(* CODESYS project PMPS.library
   Author: Alex Wallace and contributors
   Placeholder: PMPS
   Description: Collection of PMPS functionality for LCLS PLCs
   Version: 0.0.0
   DefaultNamespace: PMPS
   Title: PMPS
   Company: SLAC - LCLS

Project tree, tasks and I/O mapping:
  libraries: LCLS General, * (SLAC); Tc2_MC2, * (Beckhoff Automation GmbH); Tc2_Standard, * (Beckhoff Automation GmbH); Tc2_System, * (Beckhoff Automation GmbH); Tc2_Utilities, * (Beckhoff Automation GmbH); Tc3_JsonXml, * (Beckhoff Automation GmbH); Tc3_Module, * (Beckhoff Automation GmbH); TcUnit, * (www.tcunit.org)
  DUTs/
    InternalDUT/
      data type E_BPTMState
      data type E_MPSBeamRates
      data type K_Apertures
      data type K_Stopper
      data type L_Apertures
      data type L_Stopper
      data type ST_FF
      data type ST_FFInfo
      data type ST_FFOverride
      data type ST_PMPS_Aperture
      data type ST_PMPS_Attenuator
      data type T_HashTableEntry
    UserDUT/
      data type ST_BeamParams
      data type ST_Device
    data type ST_DeviceState
    data type ST_DeviceStateExt
    data type ST_DeviceStateTable
  GVLs/
    global variables GVL_CUSTOM_CONSTANTS
    global variables PMPS_GVL
    global variables PMPS_TOOLS
  HelperFunctions/
    TypeTranslators/
      function APT_TO_IO [ST]
      function ATT_TO_IO [ST]
      function BP_TO_IO [ST]
      function F_DeviceState_To_DeviceStateExt [ST]
      function IO_TO_APT [ST]
      function IO_TO_ATT [ST]
      function IO_TO_BP [ST]
    function F_DifferentBeamParams [ST]
    function F_eVRangeCalculator [ST]
    function F_eVWithinSpec [ST]
    function F_PMPS_JSON [ST]
    function F_SafeBPCompare [ST]
    function F_SetBeamParams [ST]
    function F_SetStateParams [ST]
  MajorComponents/
    Arbiter/
      function block FB_Arbiter [ST]: AddRequest, ArbitrateBP, CheckRequest, CheckRequestInPool, ElevateRequest, FB_init, GetArbitratedBP, RemoveRequest, RequestBP
      function block FB_BeamParamAssertionPool [ST]: A_Add, A_Count, A_GetFirst, A_GetNext, A_Lookup, A_Remove, A_Reset
    FastFaults/
      function block FB_FastFault [ST]
      function block FB_HardwareFFOutput [ST]: EvaluateOutput, EvaluateOverrides, EvaluateVetos, Execute, ExecuteLogging, FormulateLogJson, IdxCheckIn, Register
    InterPlcComm/
      function block FB_ArbiterToSubSys_IO [ST]
      function block FB_SubSysToArbiter_IO [ST]: CheckRequest, RequestBP
    PhotonEnergyInterface/
      function F_CalculatePhotonEnergy [ST]
      function block FB_AcceleratorLinks [ST]
      function block FB_Hgvpu [ST]: Init, UndAdrUpdate
      function block FB_LPhotonEnergy [ST]
      function block FB_SXU [ST]
      function block FB_UndulatorSegment [ST]
    PMPS_MPS_Interface/
      function block FB_BeamClassOutputs [ST]
      function block FB_CTLS_Outputs [ST]
      function block FB_PhotonEnergyWatcher [ST]
    SimulationFB/
      function block FB_eVSimulator [ST]
      function block FB_MachineSimulator [ST]
    Stoppers/
      function block FB_KStopper [ST]: FB_init
      function block FB_LStopper [ST]: FB_init
      function block FB_StopperWatcher [ST]
    function block BeamParameterTransitionManager [ST]: AssertFinalBP, AssertTransitionBP, AuthorizeTransition, DeauthorizeTransition, NewTarget_ENTRY, RemoveTransitionAssertion, SetNewTarget, WaitingForFinalAssertion_DO, WaitingForFinalAssertion_EXIT, WaitingForTransitionAssertion_DO, WaitingForTransitionAssertion_EXIT
    function block FB_BPControlDevice [ST]: FB_init
    function block FB_BPRequestor [ST]: CheckRequest, RequestBP
    function block FB_LinearDeviceStateTable [ST]: A_Add, A_Count, A_GetFirst, A_GetNext, A_Lookup, A_Remove, A_Reset
    function block FB_LinearGovernor [ST]
    function block FB_LRateFromEPICS [ST]
    interface I_HigherAuthority: CheckRequest, RequestBP
  TestComponents/
    data type eBPTMTestStates
    function block FB_Arbiter_Test [ST]: Arbitration, FullArbitrationStack, RequestCheckRemoveBP, StackArbiters
    function block FB_ArbToSubsys_Test [ST]: BasicFunction
    function block FB_AttenuatorSimulator [ST]
    function block FB_BPTM_Test [ST]: BPTMBasicFunction
    function block FB_DiffBP_Test [ST]: BPDiff
    function block FB_evRangeCalculator_Test [ST]: BasicFunction
    function block FB_eVWithinSpec_Test [ST]: evWithinRangeChecks
    function block FB_FastFault_Test [ST]: FFCombinedFunctionality, FFRegistration
    function block FB_PhotonEnergyWatcher_Test [ST]: PEWatcherBasicFunction
    function block FB_SafeBPCompare_Test [ST]: BeamOffIsSafe, BPComparisonCheck
    function block FB_SubsysToArb_Test [ST]: BasicFunction
  VISUs/
  program MAIN [ST]
*)

// DUTs/InternalDUT/E_BPTMState
TYPE E_BPTMState :
(
    Init := 0,
	NewTarget := 1,
    WaitingForTransitionAssertion := 2,
    WaitingForFinalAssertion := 3,
    Transitioning := 4,
    CleaningUp := 5,
	Idle := 6
);
END_TYPE

// DUTs/InternalDUT/E_MPSBeamRates

TYPE E_MPSBeamRates :
(
	MPSRateInvalid            :=  0,
    MPSRate0Hz                :=  1,
    (* Previously used 2 and 3 for single shot and burst *)
    MPSRate1Hz                :=  4,
    MPSRate10Hz               :=  5,
    MPSRate30Hz               :=  6,
    MPSRate60Hz               :=  7,
    MPSRate120Hz              :=  8,
    MPSRateUnknown            :=  9,
    MPSRateSingleShot         := 10,
    MPSRateBurstMode          := 11,
    MPSRateBurstModeNotActive := 12,
    MPSNumberOfBeamRates      := 13,
    MPSRateBurstInvalid       := 14
)UINT;
END_TYPE

// DUTs/InternalDUT/K_Apertures
{attribute 'qualified_only'}
{attribute 'strict'}
TYPE K_Apertures :
(
	SL1K0 := 1,
    SL2K0 := 2
);
END_TYPE

// DUTs/InternalDUT/K_Stopper
{attribute 'qualified_only'}
{attribute 'strict'}
TYPE K_Stopper :
(
	ST1 := 1,
    ST2 := 2
);
END_TYPE

// DUTs/InternalDUT/L_Apertures
{attribute 'qualified_only'}
{attribute 'strict'}
TYPE L_Apertures :
(
	SL1L0 := 1,
    SL2L0 := 2
);
END_TYPE

// DUTs/InternalDUT/L_Stopper
{attribute 'qualified_only'}
{attribute 'strict'}
TYPE L_Stopper :
(
	ST1L0 := 1, // ST1
    ST1L1 := 2 // ST2
);
END_TYPE

// DUTs/InternalDUT/ST_FF
TYPE ST_FF :
STRUCT
    {attribute 'pytmc' := '
        pv: Info
     '}
    Info : ST_FFInfo;
    
    {attribute 'pytmc' := '
        pv: Ovrd
     '}
    Ovrd : ST_FFOverride;
    
    {attribute 'pytmc' := '
        pv: OK
        io: i
     '}
    OK   :   BOOL; // Fault logic state
    
    FaultAck : BOOL; // Set when faulted, reset by logger.
    ClearAck : BOOL;
    
    {attribute 'pytmc' := '
        pv: BeamPermitted
        io: i
     '}
    BeamPermitted   :   BOOL; // Result of reset, veto, and fault logic, true beam off boolean
    
    {attribute 'pytmc' := '
        pv: Reset
        io: o
     '}
    Reset   :   BOOL;
    
    bsFF    :    RS;
    rtReset    :    R_TRIG;
    ftCountFault : F_TRIG;
    
END_STRUCT
END_TYPE

// DUTs/InternalDUT/ST_FFInfo

// These elements should be set at init and never changed.

TYPE ST_FFInfo :
STRUCT
    {attribute 'pytmc' := '
        pv: Path
        io: i
     '}
    sPath   :    T_MaxString; // Full PLC path to FF object
    {attribute 'pytmc' := '
        pv: Desc
        io: i
     '}
    Desc    :   T_MaxString; // Set at instantiation to a helpful description of the fast fault purpose
    {attribute 'pytmc' := '
        pv: DevName
        io: i
     '}
    DevName :   T_MaxString; // Component name, used in diagnostic to help narrow down where beam faults are coming from
    {attribute 'pytmc' := '
        pv: TypeCode
        io: i
     '}
    TypeCode    :   UINT; // Set at instantiation to fault class code

///////////////////////////////////////////
// Warning, this variable is effectively a VETO of the fast fault if set FALSE
// Do not alter the state of this variable unless you really know what you're doing.
///////////////////////////////////////////
    {attribute 'pytmc' := '
        pv: InUse
        io: i
     '}
    InUse   :   BOOL := FALSE; // If this FF is currently in-use
///////////////////////////////////////////

 
    AutoReset   :   BOOL; // Automatically clear fast fault (latching vs non-latching)
    Vetoable  : BOOL := TRUE; // Can this fast fault be masked by the veto device input?

      {attribute 'pytmc' := '
        pv: InfoString
        io: i
     '}
    InfoString : STRING;
END_STRUCT
END_TYPE

// DUTs/InternalDUT/ST_FFOverride
TYPE ST_FFOverride :
STRUCT
    {attribute 'pytmc' := '
        pv: Duration
        io: o
     '}
    Duration : UDINT; // UDINT to be compatible with ESS module.
    
    {attribute 'pytmc' := '
        pv: Activate
        io: o
     '}
    Activate : BOOL;
    
    {attribute 'pytmc' := '
        pv: Deactivate
        io: o
     '}
    Deactivate : BOOL;
    
    {attribute 'pytmc' := '
        pv: ElapsedTime
        io: i
     '}
    ElapsedTime : UDINT; // UDINT to be compatible with ESS module.
    
    {attribute 'pytmc' := '
        pv: RemainingTime
        io: i
     '}
    RemainingTime : UDINT; // UDINT to be compatible with ESS module.
    
    {attribute 'pytmc' := '
        pv: Active
        io: i
     '} 
	Active: BOOL;
    
    Timer    :   TP;
    OvrdActLogAck : BOOL;
    OvrdExpLogAck : BOOL;
    
    tOvrdActivate : R_TRIG;
    tOvrdExpiring  : F_TRIG;
END_STRUCT
END_TYPE

// DUTs/InternalDUT/ST_PMPS_Aperture
TYPE ST_PMPS_Aperture EXTENDS ST_PMPS_Aperture_IO :
STRUCT
    (*
    {attribute 'pytmc' := 'pv: Width
            io: i
            field: EGU mm'}
    Width : REAL; // distance between horizontal slits (x)
    {attribute 'pytmc' := 'pv: Height
            io: i
            field: EGU mm'}
    Height : REAL; // distance between vertical slits (y)
    
    {attribute 'pytmc' := 'pv: OK
        io: i'}
    xOK : BOOL; // status of aperture, false if error or in motion
    *)
END_STRUCT
END_TYPE

// DUTs/InternalDUT/ST_PMPS_Attenuator
TYPE ST_PMPS_Attenuator EXTENDS ST_PMPS_Attenuator_IO :
STRUCT
    (*
        {attribute 'pytmc' := 'pv: Att
            io: i
            field: EGU %
        '}
		nTran : UINT;
        {attribute 'pytmc' := 'pv: OK
            io: i
        '}
		xAttOK : UINT; // true = no errors and attenuator is stable
        *)
END_STRUCT
END_TYPE

// DUTs/InternalDUT/T_HashTableEntry
TYPE T_HashTableEntry :
STRUCT
    {attribute 'pytmc' := '
        pv: Key
        io: i
     '}
    key : DWORD := 0;
    value : PVOID := 0;
END_STRUCT
END_TYPE

// DUTs/UserDUT/ST_BeamParams
TYPE ST_BeamParams : 
    STRUCT
        (*  Requested pre-optic attenuation %  *)
		{attribute 'pytmc' := 'pv: Transmission
            io: i
            field: EGU %
        '}
		nTran : UINT := 100;
        (* Pulse-rate *)
        {attribute 'pytmc' := 'pv: Rate
            io: i
            field: EGU Hz
        '}
        nRate : UDINT := 120;
        (* Per pulse max energy (mJ) *)
        {attribute 'pytmc' := 'pv: PulseEnergy
            io: i
            field: EGU mJ
            field: DESC This beam parameter is non-op for now.
        '}
        fPP_mJ : REAL := 20;
        (* Photon energy ranges *)
        {attribute 'pytmc' := 'pv: PhotonEnergyRanges
            io: i
            field: EGU eV'}
        {attribute 'displaymode' := 'binary'}
        neVRange : WORD := 2#1111_1111_1111_1111;
        (* Beamline attenuators *)
        {attribute 'pytmc' := 'pv: AuxAtt
        io: i'}
        astAttenuators : ARRAY [1..PMPS_GVL.AUX_ATTENUATORS] OF ST_PMPS_Attenuator;
        
        (* Stoppers *)
        {attribute 'pytmc' := 'pv: ST
        io: i'}
        aStoppers : ARRAY [1..PMPS_GVL.MAX_STOPPERS] OF BOOL;
        
        (* Apertures *)
        astApertures : ARRAY [1..PMPS_GVL.MAX_APERTURES] OF ST_PMPS_Aperture;
        
        // Toggle for watchdog
        xValidToggle : BOOL;
        // Beam parameter set is valid (if readback), or acknowledged (if request)
        {attribute 'pytmc' := 'pv: Valid
        io: i'}
        xValid : BOOL;
        // Cohort index. Identifies which cohort this BP set was included in arbitration
        {attribute 'pytmc' := 'pv: Cohort
        io: i
            field: DESC Cohort inc on each arb cycle
        '}
        nCohortInt : UDINT;
    END_STRUCT
END_TYPE

// DUTs/UserDUT/ST_Device
TYPE ST_Device :
STRUCT
	//IO
	stAxis	:	AXIS_REF;
	//The following limit switches must be TRUE or high (ie. NC) to enable that direction of motion
	//The EPICS display should show an inverted indicator to communicate end of travel reached
	i_xLoLim	AT %I*	:	BOOL; //Wire normally-closed
	i_xHiLim	AT %I*	:	BOOL; //Wire normally-closed
	
	//Acuator Parameters
	lrUpperPositionLimit	:	LREAL := 10000000000; //Use in conjuntion with limit switches or set to a huge number to ignore
	lrLowerPositionLimit	:	LREAL := -10000000000; //Use in conjuntion with limit switches or set to a huge number to ignore
	
	xEnable	:	BOOL := TRUE;
	
	//Supervisory System
	
	//MPS Override
	xOverrideMPSLimits	: BOOL := FALSE; //Set true to move beyond MPS limits. Note this will trip beam off.
	
	//Status and Faults
	xClearFaults	:	BOOL;	//Rising edge tries to clear faults of all kinds
	
	xGovernorFault	:	BOOL;	//Indicates governor is faulted
	xGovernorOverridden	:	BOOL; //Indicates governor is in override mode
	xSMFault		:	BOOL;	//Indicates component state machine is faulted
	
	//Device States
	StateTable		:	FB_LinearDeviceStateTable;
	
	stTransitionState	:	ST_DeviceState; //The transition state might have non-zero beam parameters
	nSafeState			:	UDINT; //State where the device is considered safe
	nTransitionState	:	UDINT;
	
	nRequestedState	:	UDINT; //EPICS control, cleaned (checked against array limits) and deposited in nTargetState
	nTargetState	:	UDINT; //The requested state should be deposited here after cleaning
	nActiveState	:	UDINT; //The last successfully reached state
	
	
END_STRUCT
END_TYPE

// DUTs/ST_DeviceState
TYPE ST_DeviceState :
STRUCT
	
	//State name
	sStateName	:	STRING;
	nStateRef	:	UDINT; //Primary key of device state database
	
	//////////////////
	// This stuff may belong in a sub-class or something
	//Position
	rPosition	:	REAL := 0; //Center of the state
	//Tolerance
	rTolerance :	REAL := 0; //+/- amount
	//////////////////
	//Required beam parameters
	stReqBeamParam	:	ST_BeamParams;

END_STRUCT
END_TYPE

// DUTs/ST_DeviceStateExt
//Use when working with states in code
//Extended with a valid boolean to indicate the structure was loaded
//properly
TYPE ST_DeviceStateExt EXTENDS ST_DeviceState :
STRUCT
	xValid	:	BOOL := FALSE;
END_STRUCT
END_TYPE

// DUTs/ST_DeviceStateTable
TYPE ST_DeviceStateTable :
STRUCT
	iDeviceID:DINT;
	iStateID:DINT;
	rTargetPosition: REAL;
	rTolerance: REAL;
	rTransmission: REAL;
	iBeamClass : DINT;
	iPulseRate: DINT;
	rPerPulseEnergy:REAL;
	rUpper_eV: REAL;
	rLower_eV: REAL;
	rPhotonEnergy: REAL;
END_STRUCT
END_TYPE

// TestComponents/eBPTMTestStates
{attribute 'qualified_only'}
{attribute 'strict'}
TYPE eBPTMTestStates :
(
    Init := 0,
    WaitingForValidID := 50,
    WaitingForTransitionAssertion := 100,
    WaitingForFinalAssertion    := 200,
    Transitioning    := 300,
    CleaningUp    := 400,
    AnotherState := 500
);
END_TYPE

// GVLs/GVL_CUSTOM_CONSTANTS
VAR_GLOBAL CONSTANT
    MAX_FAST_FAULTS : UINT := 50; // Maximum number of fast faults that can be associated with a FFO
END_VAR

// GVLs/PMPS_GVL
{attribute 'qualified_only'}
VAR_GLOBAL
    {attribute 'pytmc' := '
        pv: @(PREFIX)RequestedBP
        archive: 1Hz monitor
    '}
    stRequestedBeamParameters    :    ST_BeamParams; //Summarized request for the line, as recognized by the line arbiter PLC
    {attribute 'pytmc' := '
        pv: @(PREFIX)CurrentBP
        archive: 1Hz monitor
    '}
    stCurrentBeamParameters    :    ST_BeamParams; //Currently active BP set, broadcast by the line arbiter PLC
    
    fbLog : FB_LogMessage:=(eSubsystem:=E_Subsystem.MPS);
END_VAR
VAR_GLOBAL RETAIN    
    // Statistics
    {attribute 'pytmc' := '
        pv: @(PREFIX)SuccessfulPreemptions
        io: i
    '}
    SuccessfulPreemption : UDINT; // Any time BPTM applies a new BP request which is confirmed
    {attribute 'pytmc' := '
        pv: @(PREFIX)AccumulatedFastFaults
        io: i
    '}
    AccumulatedFF : UDINT; // Any time a FF occurs
END_VAR
VAR_GLOBAL CONSTANT
    EXCLUDED_ASSERTION_ID    :    UDINT    := 16#FFFFFFFF; //An assertion ID that should always return "not found" in the assertion pool
    VISIBLE_TEST_VELOCITY    :    LREAL    := 10;
    FAST_TEST_VELOCITY        :    LREAL    := 100;
    MAX_DEVICE_STATES        :    UDINT    := 300;

    MAX_STOPPERS    :   UINT := 16;
    {attribute 'pytmc' := '
        pv: @(PREFIX)FullBeamCnst
        archive: 1Hz monitor
        field: DESC Full beam constant
    '}    
    cstFullBeam    :    ST_BeamParams := (
        nTran := 100,
        fPP_mJ := 1E4,
        neVRange := 2#1111_1111_1111_1111,
        nRate    := UDINT#1000000
    );
    {attribute 'pytmc' := '
        pv: @(PREFIX)SafeBeamCnst
        archive: 1Hz monitor
        field: DESC Safe beam constant
    '} 
    cstSafeBeam    :    ST_BeamParams := (
        nTran := 0,
        fPP_mJ := 0,
        neVRange := 0,
        nRate    := 0
    );
    
    cnMaxStateArrayLen : INT := 20;
    
    AUX_ATTENUATORS : UINT := 16; // Maximum # of attenuators in the PMPS
    MAX_APERTURES : UINT := 4; // Maximum # of power slits in the PMPS
    {warning disable C0228}
    DUMMY_AUX_ATT_ARRAY : ARRAY [1..PMPS_GVL.AUX_ATTENUATORS] OF ST_PMPS_Attenuator;
    {warning restore C0228}
    MAX_ASSERTIONS    :    UDINT := 20; //Maximum number of assertions permitted in the arbiter
    
    g_cBoundaries    :    INT    := 15;
    {attribute 'pytmc' := '
        pv: @(PREFIX)eVRangeHyst
        archive: 1Hz monitor
        field: DESC eV Range hystersis
        field: EGU eV
    '}
    reVHyst: REAL := 5; // 
    {attribute 'pytmc' := '
        pv: @(PREFIX)eVRangeCnst
        archive: 1Hz monitor
        field: DESC eV Range constants
        field: EGU eV
    '}
    g_areVBoundaries    :    ARRAY [0..g_cBoundaries]    OF    REAL    := [
    1E3,
    2.7E3,
    4.4E3,
    6.1E3,
    7.8E3,
    9.5E3,
    11.2E3,
    12.9E3,
    14.6E3,
    16.3E3,
    18E3,
    19.7E3,
    21.4E3,
    23.1E3,
    24.8E3,
    25E3
];


//////////////////////////
// Undulator constants
//////////////////////////
    {attribute 'pytmc' := '
		pv: @(PREFIX)L:UND:FirstSegment 
		io: i
	'}
    iLowBound_LUnd  : UDINT := 24;
    {attribute 'pytmc' := '
		pv: @(PREFIX)L:UND:LastSegment
		io: i
	'}
    iHighBound_LUnd : UDINT := 46;
    {attribute 'pytmc' := '
        pv: Period
        io: i
        field: EGU mm
    '}
    fPeriod_mm_LUnd : LREAL := 26.0;
	{attribute 'pytmc' := '
        pv: @(PREFIX)L:UND:LowK
        io: i
    '}
	fLowK_LUnd : LREAL := 0.54;
	{attribute 'pytmc' := '
        pv: @(PREFIX)L:UND:HiK
        io: i
    '}
	fHiK_LUnd : LREAL := 2.5;

END_VAR

// GVLs/PMPS_TOOLS
{attribute 'qualified_only'}
VAR_GLOBAL
	fbJson : FB_JsonSaxWriter;
END_VAR

// HelperFunctions/TypeTranslators/APT_TO_IO
FUNCTION APT_TO_IO : ST_PMPS_Aperture_IO
VAR_INPUT
    Apt : ST_PMPS_Aperture;
END_VAR
VAR
END_VAR

APT_TO_IO.Height := Apt.Height;
APT_TO_IO.Width := Apt.Width;
APT_TO_IO.xOK := Apt.xOK;

END_FUNCTION

// HelperFunctions/TypeTranslators/ATT_TO_IO
FUNCTION ATT_TO_IO : ST_PMPS_Attenuator_IO
VAR_INPUT
    Att : ST_PMPS_Attenuator;
END_VAR
VAR
END_VAR

ATT_TO_IO.nTran := Att.nTran;
ATT_TO_IO.xAttOK := Att.xAttOK;

END_FUNCTION

// HelperFunctions/TypeTranslators/BP_TO_IO
FUNCTION BP_TO_IO : ST_BeamParams_IO
VAR_INPUT
    BP : ST_BeamParams;
END_VAR
VAR
    idx : UINT := 0;
END_VAR


FOR idx := 1 TO PMPS_GVL.AUX_ATTENUATORS DO
    BP_TO_IO.astAttenuators[idx] := ATT_TO_IO(BP.astAttenuators[idx]);
END_FOR

FOR idx := 1 TO PMPS_GVL.MAX_APERTURES DO
    BP_TO_IO.astApertures[idx] := APT_TO_IO(BP.astApertures[idx]);
END_FOR

BP_TO_IO.aStoppers := BP.aStoppers;
BP_TO_IO.nTran := BP.nTran;
BP_TO_IO.fPP_mJ := BP.fPP_mJ;
BP_TO_IO.nCohortInt := ULINT_TO_UDINT(BP.nCohortInt);
BP_TO_IO.neVRange := BP.neVRange;
BP_TO_IO.nRate := BP.nRate;
BP_TO_IO.xValid := BP.xValid;
BP_TO_IO.xValidToggle := BP.xValidToggle;

END_FUNCTION

// HelperFunctions/TypeTranslators/F_DeviceState_To_DeviceStateExt
FUNCTION F_DeviceState_To_DeviceStateExt : ST_DeviceStateExt
VAR_INPUT
    stDeviceState    :    ST_DeviceState;
    xValid    :    BOOL;
END_VAR
VAR
END_VAR

F_DeviceState_To_DeviceStateExt.nStateRef := stDeviceState.nStateRef;
F_DeviceState_To_DeviceStateExt.rPosition    :=    stDeviceState.rPosition;
F_DeviceState_To_DeviceStateExt.rTolerance    :=    stDeviceState.rTolerance;
F_DeviceState_To_DeviceStateExt.sStateName    := stDeviceState.sStateName;
F_DeviceState_To_DeviceStateExt.stReqBeamParam    := stDeviceState.stReqBeamParam;
F_DeviceState_To_DeviceStateExt.xValid := xValid;

END_FUNCTION

// HelperFunctions/TypeTranslators/IO_TO_APT
FUNCTION IO_TO_APT : ST_PMPS_Aperture
VAR_INPUT
    IO : ST_PMPS_Aperture_IO;
END_VAR
VAR
END_VAR

IO_TO_APT.Height := IO.Height;
IO_TO_APT.Width := IO.Width;
IO_TO_APT.xOK := IO.xOK;

END_FUNCTION

// HelperFunctions/TypeTranslators/IO_TO_ATT
FUNCTION IO_TO_ATT : ST_PMPS_Attenuator
VAR_INPUT
    IO : ST_PMPS_Attenuator_IO;
END_VAR
VAR
END_VAR

IO_TO_ATT.nTran := IO.nTran;
IO_TO_ATT.xAttOK := IO.xAttOK;

END_FUNCTION

// HelperFunctions/TypeTranslators/IO_TO_BP
FUNCTION IO_TO_BP : ST_BeamParams
VAR_INPUT
    IO : ST_BeamParams_IO;
END_VAR
VAR
    idx : UINT;
END_VAR


FOR idx := 1 TO PMPS_GVL.AUX_ATTENUATORS DO
    IO_TO_BP.astAttenuators[idx] := IO_TO_ATT(IO.astAttenuators[idx]);
END_FOR

FOR idx := 1 TO PMPS_GVL.MAX_APERTURES DO
    IO_TO_BP.astApertures[idx] := IO_TO_APT(IO.astApertures[idx]);
END_FOR

IO_TO_BP.aStoppers := IO.aStoppers;
IO_TO_BP.nTran := IO.nTran;
IO_TO_BP.fPP_mJ := IO.fPP_mJ;
IO_TO_BP.nCohortInt := ULINT_TO_UDINT(IO.nCohortInt);
IO_TO_BP.neVRange := IO.neVRange;
IO_TO_BP.nRate := IO.nRate;
IO_TO_BP.xValid := IO.xValid;
IO_TO_BP.xValidToggle := IO.xValidToggle;

END_FUNCTION

// HelperFunctions/F_DifferentBeamParams
(*Compares BeamParam1 to BeamParam2, if any parameters of BeamParam1 are different than BeamParam2
the result will be true. *)
FUNCTION F_DifferentBeamParams : BOOL
VAR_INPUT
    BeamParam1    :    ST_BeamParams;
    BeamParam2    :    ST_BeamParams;
END_VAR
VAR
    xAttOK: BOOL := FALSE;
    xPPmjOK: BOOL := FALSE;
    xEvOK: BOOL := FALSE;
    xRateOK: BOOL := FALSE;
    xaStopper : BOOL := FALSE;
    xaAtt : BOOL := FALSE;
    xaApt : BOOL := FALSE;
    
    idx : UINT;
    
    
END_VAR

xAttOK := BeamParam1.nTran <> BeamParam2.nTran;
xPPmjOK := BeamParam1.fPP_mJ <> BeamParam2.fPP_mJ;
xEvOK := BeamParam1.neVRange <> BeamParam2.neVRange;
xRateOK     := BeamParam1.nRate <> BeamParam2.nRate;

//ast Attenuators
FOR idx:=1 TO PMPS_GVL.AUX_ATTENUATORS DO
    xaAtt S= (BeamParam1.astAttenuators[idx].nTran <> BeamParam2.astAttenuators[idx].nTran);   
END_FOR

// Stoppers
FOR idx:=1 TO PMPS_GVL.MAX_STOPPERS DO
    xaStopper S= (BeamParam1.aStoppers[idx] <> BeamParam2.aStoppers[idx]);
END_FOR

// ast Apertures
FOR idx:=1 TO PMPS_GVL.MAX_APERTURES DO
    xaApt S= (BeamParam1.astApertures[idx].Height <> BeamParam2.astApertures[idx].Height) OR
            (BeamParam1.astApertures[idx].Width <> BeamParam2.astApertures[idx].Width);
END_FOR


F_DifferentBeamParams := xAttOK OR xPPmjOK OR xEvOK OR xRateOK OR xaStopper OR xaAtt OR xaApt;

END_FUNCTION

// HelperFunctions/F_eVRangeCalculator
(*
A. Wallace 2019-8-8

Provides bit range of eV.

LastWord = 0 (Result)
----------------------------------
reV = 300 = (0000_0000_0000_0010)
reV = 301 = (0000_0000_0000_0100)

LastWord = 0000_0000_0000_0010 (Result)
----------------------------------
reV = 300 + <rHyst = (0000_0000_0000_0110)
reV = 300 + >rHyst = (0000_0000_0000_0100)

*)
FUNCTION F_eVRangeCalculator : WORD // Bit-range of current photon energy
VAR_INPUT
    reV    :    REAL; // Photon energy (keV)
    LastWord    :    WORD; // Range word of previous cycle
END_VAR
VAR
    nIndex: INT;
    RangeWord: WORD;
    rPreviousBoundary: REAL := 0;
    
    MaxEv    :    REAL := PMPS_GVL.g_areVBoundaries[PMPS_GVL.g_cBoundaries]*1000;
END_VAR


IF reV < 0 THEN F_eVRangeCalculator := 16#FFFF; RETURN; END_IF // Failsafe

FOR nIndex := 0 TO PMPS_GVL.g_cBoundaries DO
    
    // If previously active then check if it should be cleared
    IF LastWord.0 THEN 
        // Hysteresis condition
        IF (reV > MIN(PMPS_GVL.g_areVBoundaries[nIndex] + PMPS_GVL.reVHyst, MaxEv) ) OR
        (reV < MAX(rPreviousBoundary - PMPS_GVL.reVHyst, 0) ) THEN
            RangeWord.0 := 0; // If out of range of hys. mark inactive
        ELSE
            RangeWord.0 := 1;
        END_IF
    ELSE // Check if we should mark as active
        IF (reV <= PMPS_GVL.g_areVBoundaries[nIndex]) AND
        (reV > rPreviousBoundary) THEN
            RangeWord.0 := 1;
        END_IF
    END_IF
    
    // Catch if the hysteresis is set too large for the range
    IF rPreviousBoundary + PMPS_GVL.reVHyst >= PMPS_GVL.g_areVBoundaries[nIndex] THEN
        RangeWord.0 := 1; // Setting the bit true here as a failsafe
        //<TODO> Add major error or warning here
    END_IF
    
    rPreviousBoundary := PMPS_GVL.g_areVBoundaries[nIndex];
    // Shift to next bit
    RangeWord := ROR(RangeWord, 1);
    LastWord := SHR(LastWord, 1);
    
END_FOR

F_eVRangeCalculator := RangeWord;

END_FUNCTION

// HelperFunctions/F_eVWithinSpec
//reV must be within permitted range.
FUNCTION F_eVWithinSpec : BOOL
VAR_INPUT
    reV    :    REAL;    //Photon energy to check if within permitted range
    nPermittedRange    :    WORD; //Permitted range
END_VAR
VAR
    //Holding register for permitted ranges
    nPermittedRangeHolding    :    WORD; 
    //For loop counter
    nIndex    :    INT;
    // Lower boundary for range check 
    rPreviousBoundary: REAL := 0;
END_VAR

(* How this works:
The within range bool is initialized to false.
Load the word representation of ranges into a holding register.
If the bit at position zero of the holding register is true, and the input eV is
below the boundary at the index position of the boundary array, and the previous boundary
(which initializes at 0), then the within range bool is set. 
Then, we stash the upper boundary as the lower boundary for the next comparison,
and shift the holding register right, which moves the next bit to the zero position.
*)
nPermittedRangeHolding := nPermittedRange;

FOR nIndex := 0 TO PMPS_GVL.g_cBoundaries DO
        
    F_eVWithinSpec S= nPermittedRangeHolding.0 AND( 
        (reV <= PMPS_GVL.g_areVBoundaries[nIndex]*1000) AND
        (reV >= rPreviousBoundary*1000) );
        
    IF F_eVWithinSpec THEN RETURN; END_IF
    
    rPreviousBoundary := PMPS_GVL.g_areVBoundaries[nIndex];
    nPermittedRangeHolding := SHR(nPermittedRangeHolding, 1);
END_FOR

END_FUNCTION

// HelperFunctions/F_PMPS_JSON
FUNCTION F_PMPS_JSON : STRING
VAR_INPUT
	sDevName : STRING := '';
	sPath : STRING := '';
	nTypeCode : UINT := 0;
END_VAR
VAR
	
END_VAR


PMPS_TOOLS.fbJson.StartObject();
PMPS_TOOLS.fbJson.AddKey('pmps_typecode');
PMPS_TOOLS.fbJson.AddUdint(nTypeCode);
PMPS_TOOLS.fbJson.AddKey('pmps_path');
PMPS_TOOLS.fbJson.AddString(sPath);
PMPS_TOOLS.fbJson.AddKey('pmps_device_name');
PMPS_TOOLS.fbJson.AddString(sDevName);
PMPS_TOOLS.fbJson.EndObject();
F_PMPS_JSON := PMPS_TOOLS.fbJson.GetDocument();
PMPS_TOOLS.fbJson.ResetDocument();

END_FUNCTION

// HelperFunctions/F_SafeBPCompare
(*Compares BeamParam1 to BeamParam2: if the parameters of BeamParam1 are more conservative than BeamParam2
the result will be true. *)
FUNCTION F_SafeBPCompare : BOOL
VAR_INPUT
    BeamParam1    :    ST_BeamParams; //Must be more conservative than 2
    BeamParam2    :    ST_BeamParams;
END_VAR
VAR
    // Internal Attenuation OK boolean
    xAttOK: BOOL := FALSE;
    // Internal Per-pulse energy OK boolean
    xPPmjOK: BOOL := FALSE;
    // Internal photon energy OK boolean
    xEvOK: BOOL := FALSE;
    // Internal Beam Rate OK boolean
    xRateOK: BOOL;
    // Beam-rate is zero, masks all others considerations.
    xZeroRate: BOOL;
    
    idx : UINT;
    xAuxAttOK : BOOL := TRUE;
    xAuxAprtOK : BOOL := TRUE; 
END_VAR


xAttOK := BeamParam1.nTran <= BeamParam2.nTran;
xPPmjOK := BeamParam1.fPP_mJ <= BeamParam2.fPP_mJ;
xEvOK := (BeamParam1.neVRange AND BeamParam2.neVRange) = BeamParam1.neVRange;
xZeroRate    := BeamParam1.nRate = 0;
xRateOK    := BeamParam1.nRate <= BeamParam2.nRate;

FOR idx:=1 to PMPS_GVL.AUX_ATTENUATORS DO
    xAuxAttOK R= BeamParam1.astAttenuators[idx].nTran > BeamParam2.astAttenuators[idx].nTran;    
END_FOR

FOR idx:=1 to PMPS_GVL.MAX_APERTURES DO
    xAuxAprtOK R= BeamParam1.astApertures[idx].Height > BeamParam2.astApertures[idx].Height OR
    BeamParam1.astApertures[idx].Width > BeamParam2.astApertures[idx].Width;
END_FOR

F_SafeBPCompare := xZeroRate OR (xAttOK AND xPPmjOK AND xEvOK AND xRateOK AND xAuxAprtOK AND xAuxAttOK);

END_FUNCTION

// HelperFunctions/F_SetBeamParams
FUNCTION F_SetBeamParams : ST_BeamParams
VAR_INPUT
    nTran    :    UINT := 0;
    fPP_mJ: REAL := 0;
    neVRange    :    WORD := 0;
    nRate    :    UDINT := 0;
    astAuxAtt : ARRAY [1..PMPS_GVL.AUX_ATTENUATORS] OF ST_PMPS_Attenuator;
END_VAR
VAR
    BeamParams    :    ST_BeamParams;
    
END_VAR

BeamParams.nTran := LIMIT(0,nTran,100);
BeamParams.astAttenuators := astAuxAtt;
BeamParams.fPP_mJ := LIMIT(0,fPP_mJ,20);
BeamParams.neVRange := neVRange;
BeamParams.nRate    := MIN(nRate,1000000);

F_SetBeamParams    := BeamParams;

END_FUNCTION

// HelperFunctions/F_SetStateParams
FUNCTION F_SetStateParams : BOOL;
VAR_INPUT
    nStateRef    :    UDINT;
    rPosition    :    REAL;
    rTolerance: REAL;
    stBeamParams    :    ST_BeamParams;
END_VAR
VAR_IN_OUT
    Table    :    FB_LinearDeviceStateTable;
END_VAR
VAR
    stDeviceState    :    ST_DeviceState;
    
END_VAR

stDeviceState.nStateRef := nStateRef;
stDeviceState.rPosition := rPosition;
stDeviceState.rTolerance := rTolerance;
stDeviceState.stReqBeamParam := stBeamParams;

Table.A_Add(
    key := nStateRef,
    putValue := stDeviceState
);

F_SetStateParams := Table.bOk;

END_FUNCTION

// MajorComponents/FB_LinearDeviceStateTable
(* This function block implements simple database. Data element values are stored in the hash table.  *)
FUNCTION_BLOCK FB_LinearDeviceStateTable
VAR_INPUT
    key         : DWORD := 0;(* Entry key: used by A_Lookup, A_Remove method, the key variable is also used by A_Add method *)
    putPosPtr    : POINTER TO T_HashTableEntry := 0;(* Hash table entry position pointer (used by A_Find, A_GetNext, A_GetPrev) *)
    putValue     : ST_DeviceState;(* Hash table entry value (used by A_AddHead, A_AddTail, A_Find )*)
END_VAR
VAR_OUTPUT
    bOk            : BOOL := FALSE;(* TRUE = Success, FALSE = Failed *)
    getPosPtr    : POINTER TO T_HashTableEntry := 0;(* Returned hash table entry position pointer *)
    getValue     : ST_DeviceState;(* Returned hash table entry value *)
    nCount        : UDINT := 0;(* Hash table size (number of used entries, used by A_Count) *)
END_VAR
VAR
    dataPool    : ARRAY[0..PMPS_GVL.MAX_DEVICE_STATES] OF ST_DeviceState;(* Structured data element pool *)
    entries        : ARRAY[0..PMPS_GVL.MAX_DEVICE_STATES] OF T_HashTableEntry;(* Max. number of hash table entries. The value of table entry = 32 bit integer (pointer to dataPool-array-entry) *)
    fbTable     : FB_HashTableCtrl;(* basic hash table control function block *)
    hTable         : T_HHASHTABLE;(* hash table handle *)
    pRefPtr        : POINTER TO ST_DeviceState := 0;
    indexOfElem    : ULINT;(* Integer value (max. size: x86=>32bit, x64=>64bit)*)
END_VAR

;

ACTION A_Add:
(* Adds entry to the table *)
MEMSET( ADR( getValue ), 0, SIZEOF( getValue ) );
getPosPtr := 0;

fbTable.A_Add( hTable := hTable, key := key, putValue := ADR(PMPS_GVL.cstSafeBeam)(* we will set this value later *), getPosPtr=>getPosPtr, bOk=>bOk );(* Add new element to the table, getPosPtr points to the new entry *)
IF fbTable.bOk THEN(* Success *)
    fbTable.A_GetIndexAtPosPtr( hTable := hTable, putPosPtr := getPosPtr, getValue =>indexOfElem, bOk=>bOk );(* Get array index of getPosPtr entry *)
    IF fbTable.bOk THEN(* Success *)
        pRefPtr     := ADR( dataPool[indexOfElem] );(* Get pointer to the data element *)

        pRefPtr^ := putValue;(* copy application value *)

        fbTable.A_Add( hTable := hTable, key := key, putValue := pRefPtr, bOk=>bOk );(* Assign the entry value = pointer to the data element *)
        IF fbTable.bOk THEN(* Success *)
            getValue := putValue;
        END_IF
    END_IF
END_IF
END_ACTION

ACTION A_Count:
(* Count number of used entries *)
nCount := hTable.nCount;
bOk := TRUE;
END_ACTION

ACTION A_GetFirst:
(* Get first entry position pointer and value *)
MEMSET( ADR( getValue ), 0, SIZEOF( getValue ) );
getPosPtr := 0;

fbTable.A_GetFirst( hTable := hTable, putPosPtr := putPosPtr, getValue=>pRefPtr, getPosPtr=>getPosPtr, bOk=>bOk );
IF fbTable.bOk THEN
    getValue := pRefPtr^;
END_IF
END_ACTION

ACTION A_GetNext:
(* Get next entry position pointer and value *)
MEMSET( ADR( getValue ), 0, SIZEOF( getValue ) );
getPosPtr := 0;
bOk := FALSE;

IF putPosPtr = 0 THEN
    RETURN;
END_IF

fbTable.A_GetNext( hTable := hTable, putPosPtr := putPosPtr, getValue=>pRefPtr, getPosPtr=>getPosPtr, bOk=>bOk );
IF fbTable.bOk THEN
    getValue := pRefPtr^;
END_IF
END_ACTION

ACTION A_Lookup:
(* Lookup for entry by key  *)
MEMSET( ADR( getValue ), 0, SIZEOF( getValue ) );
getPosPtr := 0;

fbTable.A_Lookup( key := key, hTable := hTable, putPosPtr := putPosPtr, getValue=>pRefPtr, getPosPtr=>getPosPtr, bOk=>bOk );
IF fbTable.bOk THEN
    getValue := pRefPtr^;
END_IF
END_ACTION

ACTION A_Remove:
(* Search for entry and remove it *)
MEMSET( ADR( getValue ), 0, SIZEOF( getValue ) );
getPosPtr := 0;

fbTable.A_Remove( key := key, hTable := hTable, putPosPtr := putPosPtr, getValue=>pRefPtr, getPosPtr=>getPosPtr, bOk=>bOk );
IF fbTable.bOk THEN
    getValue := pRefPtr^;
END_IF
END_ACTION

ACTION A_Reset:
(* Reset/initialize linked list *)
MEMSET( ADR( getValue ), 0, SIZEOF( getValue ) );
getPosPtr := 0;
bOk := F_CreateHashTableHnd( ADR( entries ), SIZEOF( entries ), hTable );(* Intialize table handle *)
fbTable.A_Reset( hTable := hTable, bOk=>bOk );
nCount := 0;
END_ACTION

END_FUNCTION_BLOCK

// MajorComponents/Arbiter/FB_Arbiter
(* FB Arbiter
A. Wallace 2020-6-26

The arbiter primary objectives are:
- Provide a simple interface for devices to request beam parameter sets
- Provide a way for devices to verify their BPS is active in the arbiter
- Provide a way for devices remove their requests from evaluation
- Evaluate all active beam parameter requests registered with the aribiter,
to determine the safest combination of all sets, provide this set as an output.
- Do all of this with minimal overhead

To these ends, the arbiter uses a hash-table, the rows being a state-id as the key, and a corresponding
 beam parameter set to be evaluated against all the other sets (or rows), in the table.
 
The hash table can be thought of as an array on steriods, they are worth reading about, suffice to say
the hash table will tell you when you reach the end of all the entries, and enables us to find entries quickly.

These features efficiently address the addition, removal, and verification of beam parameter sets listed in the above requirements.
*)

FUNCTION_BLOCK FB_Arbiter IMPLEMENTS I_HigherAuthority
VAR_INPUT
END_VAR
VAR_OUTPUT
    {attribute 'pytmc' := '
        pv: ArbitratedBP
        io: i
        field: DESC Arbitrated BP
     '}
    q_stBeamParams    :    ST_BeamParams; //Updated on each cycle of the arbiter FB with the current arbitrated beam parameter set
    
    q_xStateIDFound    :    BOOL; //Set true if a state-id is found in the assertion pool after calling A_VerifyAssertion
END_VAR
VAR
    {attribute 'pytmc' := '
        pv: AP
        io: i
        field: DESC Assertion Pool
     '}
    fbBPAssertionPool    :    FB_BeamParamAssertionPool; //Table of active beam parameter assertions

    xRequestMade : BOOL; // Arbiter has confirmed its request has made it into the beam parameter request    
    
    {attribute 'pytmc' := '
        pv: ArbiterID
        io: i
        field: DESC Arbiter ID for elev. req.
     '}
    nArbiterID : UDINT; // Arbiter ID, used for making higher-level BP requests
    {attribute 'pytmc' := '
        pv: CohortCounter
        io: i
        field: DESC Intrnl cohort counter
     '}
    nArbiterCohort : UDINT := 1; // The cohort index keeps track of which beam parameter requests have been included in higher-level arbitrations
    // Init to 1, provides a guard against default cohort value in BP requests.
    {attribute 'pytmc' := '
        pv: ActiveInArbitration
        io: i
        field: DESC True if this arbiter's req is included
     '}
    xActiveInArbitration : BOOL; // True when this arbiter's request is included in all higher-level arbitrations
	
	nEntryCount : UDINT;
END_VAR

// Adds a request to the arbiter pool.
// Returns true if the request was successfully added, false if not enough space or a request with the same ID is already present.
METHOD AddRequest : BOOL
VAR_INPUT
    nReqID    :    DWORD; // Unique ID within aribter for the request. Make sure this is unique for every device + state combination
    stReqBP        :    ST_BeamParams; //Requested beam params
END_VAR
VAR_INST
    fbLog : FB_LogMessage;
END_VAR
// If the request is already in the pool, then skip the rest.
// This is flawed, needs to update the request if it's already in the pool, despite having the same ID
IF THIS^.CheckRequestInPool(nReqID) THEN
    AddRequest := FALSE;
    RETURN;
END_IF

IF nReqID <> PMPS_GVL.EXCLUDED_ASSERTION_ID THEN
    stReqBP.nCohortInt := nArbiterCohort; // Set the cohort number for this BP request.
    
    THIS^.fbBPAssertionPool.A_Add(
        key := nReqID,
        putValue := stReqBP
    );
END_IF
    
IF NOT THIS^.fbBPAssertionPool.bOk THEN
    fbLog(sMsg:=CONCAT(DWORD_TO_STRING(nReqID),'Addition to arbiter assertion pool failed'),
            eSevr:=TcEventSeverity.Warning,
            eSubsystem:=E_Subsystem.MPS);
ELSIF THIS^.fbBPAssertionPool.bOk THEN
	fbLog(sMsg:=CONCAT(DWORD_TO_STRING(nReqID),'Added to pool'),
            eSevr:=TcEventSeverity.Verbose,
            eSubsystem:=E_Subsystem.MPS);
END_IF

// With any new request reset the internal arbiter "done" flag
xRequestMade R= THIS^.fbBPAssertionPool.bOk;

AddRequest := THIS^.fbBPAssertionPool.bOk;
END_METHOD

// Kernel of the arbiter
// Logic for determining which beam parameter is the most conservative across all request sets.
METHOD INTERNAL ArbitrateBP : ST_BeamParams
VAR_INPUT
    stBP1    :    ST_BeamParams;
    stBP2    :    ST_BeamParams;
END_VAR
VAR
    idx : UINT := 1;
END_VAR
//<TODO>Add something here to register the key that won for each param

//Attenuation
ArbitrateBP.nTran := MIN(stBP1.nTran, stBP2.nTran);

FOR idx := 1 TO PMPS_GVL.AUX_ATTENUATORS DO
    ArbitrateBP.astAttenuators[idx].nTran := MIN(stBP1.astAttenuators[idx].nTran, stBP2.astAttenuators[idx].nTran);
END_FOR

//Apertures
FOR idx := 1 TO PMPS_GVL.MAX_APERTURES DO
    ArbitrateBP.astApertures[idx].Height := MIN(stBP1.astApertures[idx].Height, stBP2.astApertures[idx].Height);
    ArbitrateBP.astApertures[idx].Width := MIN(stBP1.astApertures[idx].Width, stBP2.astApertures[idx].Width);
END_FOR

//Pulse energy
ArbitrateBP.fPP_mJ := MIN(stBP1.fPP_mJ, stBP2.fPP_mJ);

//Photon energy ranges
ArbitrateBP.neVRange := stBP1.neVRange AND stBP2.neVRange;

//Rate
ArbitrateBP.nRate := MIN(stBP1.nRate, stBP2.nRate);
END_METHOD

(* Checks request ID is included in arbitration all the way to the accelerator interface
Use like so:
IF fbArbiter.CheckRequest(nStateIDAssertionToCheck) AND (other logic) THEN:
    Request is found and active in arbitration,. Do something.
ELSE:
    Request was not found, or is not yet included in arbitration. Don't do something/ wait.

*)
METHOD CheckRequest : BOOL
VAR_INPUT
    nReqID    :    DWORD;
END_VAR
VAR
    BP : ST_BeamParams;
END_VAR
fbBPAssertionPool.A_Lookup(key := nReqID);

// Verify BP is acknowledged
BP := fbBPAssertionPool.getValue;

// This logic:
// Did we find the assertion in the pool?
// Is the assertion cohort number less than the current cohort and greater than zero?
// Is the Aribter itself active in arbitration?
CheckRequest := fbBPAssertionPool.bOk AND 
                BP.nCohortInt < nArbiterCohort AND
                BP.nCohortInt > 0 AND 
                xActiveInArbitration;
END_METHOD

// Verify request is at least in the local arbiter
// Does not verify request has been included in arbitration.
// Use CheckRequest instead.
METHOD CheckRequestInPool : BOOL
VAR_INPUT
    nReqID    :    DWORD;
END_VAR
THIS^.fbBPAssertionPool.A_Lookup(key := nReqID);

CheckRequestInPool := THIS^.fbBPAssertionPool.bOk;
END_METHOD

// <Arbiter Internal>
// Elevates the arbitrated BP set to something above.
// Could be another arbiter, or a BP requester/ IO, 
// or an FB that locks in a specific portion of the BP set.
METHOD ElevateRequest : BOOL 
VAR_INPUT
    HigherAuthority : I_HigherAuthority;
END_VAR
(*
This method should only be used with one higher level component.
*)

IF NOT xRequestMade THEN
    xRequestMade := HigherAuthority.RequestBP(nReqID := nArbiterID, stReqBP := GetArbitratedBP());
    xActiveInArbitration := FALSE;
END_IF

IF HigherAuthority.CheckRequest(nReqID := nArbiterID) AND NOT xActiveInArbitration THEN // Check request must verify the ID is present and accounted for in arbitration
    nArbiterCohort := nArbiterCohort + 1; // This cohort number is for all subordinate requests within the arbiter
    xActiveInArbitration := TRUE;
END_IF
END_METHOD

METHOD FB_init : BOOL
VAR_INPUT
	bInitRetains : BOOL; // if TRUE, the retain variables are initialized (warm start / cold start)
	bInCopyCode : BOOL;  // if TRUE, the instance afterwards gets moved into the copy code (online change)
    nID : DWORD := PMPS_GVL.EXCLUDED_ASSERTION_ID; // Arbiter ID, must be globally unique.
END_VAR
nArbiterID := nId;
fbBPAssertionPool.A_Reset();
END_METHOD

// Executes Arbitration between all requested beam parameter sets
METHOD INTERNAL GetArbitratedBP : ST_BeamParams
VAR_INPUT
END_VAR
VAR
    getPosPtr    : POINTER TO T_HashTableEntry := 0;
    getBPStruct    :    ST_BeamParams;
    
    stOutputBP    :    ST_BeamParams; //Holding struct for arbitration process
END_VAR
VAR_INST
    xFirstPass : BOOL := TRUE;
    fbGetCurTaskIdx : GETCURTASKINDEX;
    LastCycleCount : UDINT;
    fbLogMessage : FB_LogMessage;
END_VAR
//Arbitrate
(*
This step cycles through every hash table entry, comparing
the beam parameters from each assertion to what we're planning
to assert.

The safer of the two parameters is kept so at the end we may
have a mix of beam parameters, the composition being safe for
all asserters.

*)

THIS^.fbBPAssertionPool.A_GetFirst( putPosPtr := 0, getPosPtr=>getPosPtr, getValue=>getBPStruct );
IF THIS^.fbBPAssertionPool.bOk THEN //If the table is empty (not OK), we are left with the default stOutputBP set above.
    
    //The first entry in the hash table is taken as the setting to arbitrate against
    stOutputBP := F_SetBeamParams(
        nTran := getBPStruct.nTran,
        astAuxAtt := getBPStruct.astAttenuators,
        fPP_mJ := getBPStruct.fPP_mJ,
        neVRange    := getBPStruct.neVRange,
        nRate := getBPStruct.nRate
    );

    REPEAT
        THIS^.fbBPAssertionPool.A_GetNext( putPosPtr := THIS^.fbBPAssertionPool.getPosPtr, getPosPtr=>getPosPtr, getValue=>getBPStruct );
        IF THIS^.fbBPAssertionPool.bOk THEN
            stOutputBP := ArbitrateBP(stOutputBP, getBPStruct);
        END_IF
    UNTIL NOT fbBPAssertionPool.bOk
    END_REPEAT
ELSE
    //Full beam if there are no arbitration requests
    stOutputBP := PMPS_GVL.cstFullBeam;
END_IF
(*
stOutputBP.AckInt := stOutputBP.AckInt + 1; // Arbitration cycle

// Verify this function hasn't been run twice this cycle
IF xFirstPass THEN
    fbGetCurTaskIdx();
END_IF

IF LastCycleCount <> _TaskInfo[fbGetCurTaskIdx.index].CycleCount THEN
    // Good
    LastCycleCount := _TaskInfo[fbGetCurTaskIdx.index].CycleCount;
ELSE
    fbLogMessage(i_sMsg := 'GetArbitratedBP run more than once in a cycle.',
        i_eSevr := E_MesgSevr.Error,
        i_eSubsystem := E_Subsystem.MPS);
END_IF
*)


q_stBeamParams := stOutputBP;

GetArbitratedBP := stOutputBP;

GetArbitratedBP.xValidToggle := NOT GetArbitratedBP.xValidToggle;

fbBPAssertionPool.A_Count();
IF fbBPAssertionPool.bOk THEN
	nEntryCount := fbBPAssertionPool.nCount ;
END_IF

xFirstPass := FALSE;
END_METHOD

(* Removes request from abritration. *)
METHOD RemoveRequest : BOOL
VAR_INPUT
    nReqId    :    DWORD;
END_VAR
VAR_INST
    fbLog : FB_LogMessage;
END_VAR
IF nReqId <> PMPS_GVL.EXCLUDED_ASSERTION_ID THEN
    THIS^.fbBPAssertionPool.A_Remove(key := nReqId);
    
    IF THIS^.fbBPAssertionPool.bOk THEN
        	(*fbLog(sMsg:=CONCAT(DWORD_TO_STRING(nReqID),'Removed from pool'),
            eSevr:=TcEventSeverity.Verbose,
            eSubsystem:=E_Subsystem.MPS);*)
    ELSE
        (*fbLog(sMsg:=CONCAT(DWORD_TO_STRING(nReqID),'Failed to remove from pool'),
            eSevr:=TcEventSeverity.Warning,
            eSubsystem:=E_Subsystem.MPS);*)
    END_IF
END_IF

// With any new request reset the internal arbiter "done" flag
xRequestMade R= THIS^.fbBPAssertionPool.bOk;

RemoveRequest := THIS^.fbBPAssertionPool.bOk;
END_METHOD

METHOD RequestBP : BOOL
VAR_INPUT
	(*StateID of state requesting beam parameter set*)
	nReqID	: DWORD;
	(*Requested beam params*)
	stReqBP	: ST_BeamParams;
END_VAR
RequestBP := AddRequest(nReqID := nReqID, stReqBP := stReqBP);
END_METHOD

END_FUNCTION_BLOCK

// MajorComponents/I_HigherAuthority
INTERFACE I_HigherAuthority

METHOD CheckRequest : BOOL
VAR_INPUT
    nReqID    :    DWORD;
END_VAR
END_METHOD

METHOD RequestBP : BOOL
VAR_INPUT
    nReqID    :    DWORD; //StateID of state requesting beam parameter set
    stReqBP        :    ST_BeamParams; //Requested beam params
END_VAR
END_METHOD

END_INTERFACE

// MajorComponents/Arbiter/FB_BeamParamAssertionPool
(* This function block implements simple database. Data element values are stored in the hash table.  *)
FUNCTION_BLOCK FB_BeamParamAssertionPool
VAR_INPUT
    key         : DWORD := 0;(* Entry key: used by A_Lookup, A_Remove method, the key variable is also used by A_Add method *)
    putPosPtr    : POINTER TO T_HashTableEntry := 0;(* Hash table entry position pointer (used by A_Find, A_GetNext, A_GetPrev) *)
    putValue     : ST_BeamParams;(* Hash table entry value (used by A_AddHead, A_AddTail, A_Find )*)
END_VAR
VAR_OUTPUT
    bOk            : BOOL := FALSE;(* TRUE = Success, FALSE = Failed *)
    getPosPtr    : POINTER TO T_HashTableEntry := 0;(* Returned hash table entry position pointer *)
    getValue     : ST_BeamParams;(* Returned hash table entry value *)
    nCount        : UDINT := 0;(* Hash table size (number of used entries, used by A_Count) *)
END_VAR
VAR
    {attribute 'pytmc' := '
        pv: Entry
        io: i
     '}
    dataPool    : ARRAY[0..PMPS_GVL.MAX_ASSERTIONS] OF ST_BeamParams;(* Structured data element pool *)
    {attribute 'pytmc' := '
        pv: Key
        io: i
     '}
    entries        : ARRAY[0..PMPS_GVL.MAX_ASSERTIONS] OF T_HashTableEntry;(* Max. number of hash table entries. The value of table entry = 32 bit integer (pointer to dataPool-array-entry) *)
    fbTable     : FB_HashTableCtrl;(* basic hash table control function block *)
    hTable         : T_HHASHTABLE;(* hash table handle *)
    pRefPtr        : POINTER TO ST_BeamParams := 0;
    indexOfElem    : ULINT;(* Integer value (max. size: x86=>32bit, x64=>64bit)*)
END_VAR

;

ACTION A_Add:
(* Adds entry to the table *)
MEMSET( ADR( getValue ), 0, SIZEOF( getValue ) );
getPosPtr := 0;

fbTable.A_Add( hTable := hTable, key := key, putValue := ADR(PMPS_GVL.cstSafeBeam)(* we will set this value later *), getPosPtr=>getPosPtr, bOk=>bOk );(* Add new element to the table, getPosPtr points to the new entry *)
IF fbTable.bOk THEN(* Success *)
    fbTable.A_GetIndexAtPosPtr( hTable := hTable, putPosPtr := getPosPtr, getValue =>indexOfElem, bOk=>bOk );(* Get array index of getPosPtr entry *)
    IF fbTable.bOk THEN(* Success *)
        pRefPtr     := ADR( dataPool[indexOfElem] );(* Get pointer to the data element *)

        pRefPtr^ := putValue;(* copy application value *)

        fbTable.A_Add( hTable := hTable, key := key, putValue := pRefPtr, bOk=>bOk );(* Assign the entry value = pointer to the data element *)
        IF fbTable.bOk THEN(* Success *)
            getValue := putValue;
        END_IF
    END_IF
END_IF
END_ACTION

ACTION A_Count:
(* Count number of used entries *)
nCount := hTable.nCount;
bOk := TRUE;
END_ACTION

ACTION A_GetFirst:
(* Get first entry position pointer and value *)
MEMSET( ADR( getValue ), 0, SIZEOF( getValue ) );
getPosPtr := 0;

fbTable.A_GetFirst( hTable := hTable, putPosPtr := putPosPtr, getValue=>pRefPtr, getPosPtr=>getPosPtr, bOk=>bOk );
IF fbTable.bOk THEN
    getValue := pRefPtr^;
END_IF
END_ACTION

ACTION A_GetNext:
(* Get next entry position pointer and value *)
MEMSET( ADR( getValue ), 0, SIZEOF( getValue ) );
getPosPtr := 0;
bOk := FALSE;

IF putPosPtr = 0 THEN
    RETURN;
END_IF

fbTable.A_GetNext( hTable := hTable, putPosPtr := putPosPtr, getValue=>pRefPtr, getPosPtr=>getPosPtr, bOk=>bOk );
IF fbTable.bOk THEN
    getValue := pRefPtr^;
END_IF
END_ACTION

ACTION A_Lookup:
(* Lookup for entry by key  *)
MEMSET( ADR( getValue ), 0, SIZEOF( getValue ) );
getPosPtr := 0;

fbTable.A_Lookup( key := key, hTable := hTable, putPosPtr := putPosPtr, getValue=>pRefPtr, getPosPtr=>getPosPtr, bOk=>bOk );
IF fbTable.bOk THEN
    getValue := pRefPtr^;
END_IF
END_ACTION

ACTION A_Remove:
(* Search for entry and remove it *)
MEMSET( ADR( getValue ), 0, SIZEOF( getValue ) );
getPosPtr := 0;

fbTable.A_Remove( key := key, hTable := hTable, putPosPtr := putPosPtr, getValue=>pRefPtr, getPosPtr=>getPosPtr, bOk=>bOk );
IF fbTable.bOk THEN
    getValue := pRefPtr^;
END_IF
END_ACTION

ACTION A_Reset:
(* Reset/initialize linked list *)
MEMSET( ADR( getValue ), 0, SIZEOF( getValue ) );
getPosPtr := 0;
bOk := F_CreateHashTableHnd( ADR( entries ), SIZEOF( entries ), hTable );(* Intialize table handle *)
fbTable.A_Reset( hTable := hTable, bOk=>bOk );
nCount := 0;
END_ACTION

END_FUNCTION_BLOCK

// MajorComponents/FastFaults/FB_FastFault
(* Fast Fault
2019-9-13 A. Wallace

Use this block to generate a beam-off fault. Connects to a fast fault hardware output 
function block to contribute to the state of the fast fault output (FFO).

If the i_xOK goes false, the associated FFO will go false, despite the state of any other
contributing fast faults, unless the FFO is currently vetoed.

*)
{attribute 'reflection'}
FUNCTION_BLOCK FB_FastFault
VAR_INPUT

    i_xOK        :    BOOL; // Connect to fast-fault condition (false produces fault)
    i_xReset    :    BOOL; // Resets when i_xOK is true and this is true
    i_xAutoReset : BOOL := FALSE; // Automatically clear fast fault (latching vs non-latching)
    i_xVetoable : BOOL := TRUE; // Mask this fast fault if the FFO veto device is true
    
    i_DevName : T_MaxString := ''; // Device name for diagnostic
    i_Desc : T_MaxString := ''; // Description of fast fault (you should set at init)
    i_TypeCode : UINT; // Error code for classifying fast faults
END_VAR
VAR_OUTPUT
    o_xFFLine    :    BOOL; //Connect to HW output or another FF input if you like (Optional)
END_VAR
VAR_IN_OUT
    io_fbFFHWO        :    FB_HardwareFFOutput; //Point to FB_HardwareFFOutput of your choice
END_VAR
VAR
    {attribute 'instance-path'}
    {attribute 'noinit'}
    sPath    :    T_MaxString;
    
    FFInfo : ST_FFInfo;
    
    RegistrationIdx : UINT := 1; // The index this FF was registered in the FFO
    
    xInit    :    BOOL :=TRUE;
    
    InfoStringFmtr : FB_FormatString;
    
    InUse : T_MaxString;
    AutoReset : T_MaxString;

END_VAR

IF xInit    THEN
    FFInfo.sPath := sPath;
    FFInfo.InUse := True;
    FFInfo.TypeCode := i_TypeCode;
    FFInfo.DevName := i_DevName;
    FFInfo.Desc := i_Desc;
    FFInfo.AutoReset := i_xAutoReset;
    FFInfo.Vetoable := i_xVetoable;
    
    InUse := BOOL_TO_STRING(FFInfo.InUse);
    AutoReset := BOOL_TO_STRING(FFInfo.AutoReset);
    InfoStringFmtr(sFormat:='%s;%s;%X;%s;%s;%s;',
        arg1 := F_STRING(FFinfo.sPath),
        arg2 := F_STRING(InUse),
        arg3 := F_WORD(FFInfo.TypeCode),
        arg4 := F_STRING(FFInfo.DevName),
        arg5 := F_STRING(FFInfo.Desc),
        arg6 := F_STRING(AutoReset),
        sOut=>FFInfo.InfoString);
    io_fbFFHWO.Register(
        stFFInfo:=FFInfo, 
        Idx=>RegistrationIdx);
    //<TODO> if registration doesn't succeed, send warning to diagnostic
    xInit := FALSE;
END_IF

io_fbFFHWO.IdxCheckIn(Idx:=RegistrationIdx, OK := i_xOK, Reset:= i_xReset);

END_FUNCTION_BLOCK

// MajorComponents/FastFaults/FB_HardwareFFOutput
{attribute 'reflection'}
FUNCTION_BLOCK FB_HardwareFFOutput
VAR CONSTANT
    FF_ARRAY_UPPER_BOUND : DINT := MAX_FAST_FAULTS;
END_VAR
VAR_INPUT
    {attribute 'pytmc' := '
        pv: ClearFault
        io: o
        field: DESC Might be overidden by PLC writes
     '}
    i_xReset    :    BOOL;
    {attribute 'pytmc' := '
        pv: EnableVeto
        io: o
     '}
    i_xVeto    :    BOOL;
    bAutoReset : BOOL := FALSE; // Set true for the FFO to automatically permit beam again after all fast faults are cleared
END_VAR
VAR_OUTPUT
    {attribute 'pytmc' := '
        pv: FaultHWO
        io: i
        field: DESC Hardware Output Status
     '}
    q_xFastFaultOut    AT %Q*    :    BOOL;
END_VAR
VAR_IN_OUT

END_VAR
VAR
    {attribute 'pytmc' := '
        pv: FF
     '}
    astFF : ARRAY[1..FF_ARRAY_UPPER_BOUND] OF ST_FF;
    
    {attribute 'pytmc' := '
        pv: RegistrationFailure
        io: io
     '}
    xFastFaultRegFail  :   BOOL := FALSE; // Set true if a fast fault fails to register. Holds beam off.
    tFFRegFail : F_TRIG;
    
    {attribute 'instance-path'}
    {attribute 'noinit'}
    sPath    :    T_MaxString;

	{attribute 'pytmc' := '
        pv: OK
        io: i
     '}
    xOK    :    BOOL:= TRUE; // Current internal state of FFO, indicates if FFO will accept a reset
    
    rtReset    :    R_TRIG;
    rtResetandOK : R_TRIG;
    
    nIndex    :    UINT := 1;
	
	IdxOK: BOOL;
    
    
    fbJson : FB_JsonSaxWriter;
    pmpsTypeCode : UDINT := 0; // shows up in json as pmps_typecode
    fbLogger : FB_LogMessage := (
        eSevr := TcEventSeverity.Critical,
        eSubsystem := E_Subsystem.MPS);

END_VAR

// <TODO> latch off beam if DI card status goes bad

ACTION EvaluateOutput:

////////////////////////////////////////////////////////////////
// Critical code. Do not touch unless you know what you're doing
////////////////////////////////////////////////////////////////

//<TODO> add diagnostic for success or failure of reset
rtReset(CLK:=i_xReset);
rtResetandOK(CLK:=(rtReset.Q OR bAutoReset) AND xOK);

q_xFastFaultOut S= rtResetandOK.Q;
q_xFastFaultOut R= (NOT xOK OR xFastFaultRegFail);

//Reset OK for next cycle
xOK := True;

////////////////////////////////////////////////////////////////
END_ACTION

METHOD EvaluateOverrides : BOOL
VAR_INPUT
END_VAR
VAR
    FF : REFERENCE TO ST_FF;
    EvalIdx: DINT := 1;
END_VAR

FOR EvalIdx := 1 TO FF_ARRAY_UPPER_BOUND DO
    
    FF REF= astFF[EvalIdx];
    
    IF NOT FF.Info.InUse THEN 
        CONTINUE;
    ELSE
        // Veto timer
        IF FF.Ovrd.Deactivate THEN 
            FF.Ovrd.Timer.PT := T#0s; // Only needs to be set zero for one cycle
        ELSE
            FF.Ovrd.Timer.PT := UDINT_TO_TIME(FF.Ovrd.Duration);
        END_IF
        
        // UDINT conversions for ESS module compatibility.
        FF.Ovrd.Timer(
            IN := FF.Ovrd.Activate, // Rising edge activated
            Q => FF.Ovrd.Active);
            
        FF.Ovrd.tOvrdActivate(CLK:=FF.Ovrd.Active);
        FF.Ovrd.OvrdActLogAck S= FF.Ovrd.tOvrdActivate.Q;
        
        FF.Ovrd.tOvrdExpiring(CLK:=FF.Ovrd.Active);
        FF.Ovrd.OvrdExpLogAck S= FF.Ovrd.tOvrdExpiring.Q;
            
        FF.Ovrd.ElapsedTime := TIME_TO_UDINT(FF.Ovrd.Timer.ET);
        
        FF.Ovrd.RemainingTime := MAX(0, FF.Ovrd.Duration - FF.Ovrd.ElapsedTime);
        
        // Clear pushbuttons
        FF.Ovrd.Activate := FALSE;
        FF.Ovrd.Deactivate := FALSE;
        
    END_IF    
END_FOR
END_METHOD

{attribute 'obsolete' := 'Use EvaluateOverrides instead.'} 
METHOD EvaluateVetos : BOOL
VAR_INPUT
END_VAR
END_METHOD

ACTION Execute:
EvaluateOutput();
EvaluateOverrides();
ExecuteLogging();
END_ACTION

METHOD ExecuteLogging : BOOL
VAR_INPUT
END_VAR
VAR
    FF : REFERENCE TO ST_FF;
    logIdx : DINT := 1; 
END_VAR
VAR_INST
    HelloTimer : TOF := ( PT:=T#24h );
END_VAR

FOR logIdx := 1 to FF_ARRAY_UPPER_BOUND do
    
    FF REF= astFF[logIdx];
    
    IF NOT FF.Info.InUse THEN 
        CONTINUE;
    ELSE
        IF FF.FaultAck THEN

            pmpsTypeCode := 1;
            FormulateLogJson(FF);
            fbLogger(sMsg := 'Fault, beam off', eSevr:=TcEventSeverity.Critical);
            
            FF.FaultAck := FALSE;
        END_IF
        
        IF FF.Ovrd.OvrdActLogAck THEN
            
            pmpsTypeCode := 2;
            FormulateLogJson(FF);
            
            fbLogger(sMsg := 'Override activated', eSevr:=TcEventSeverity.Warning);
            
            FF.Ovrd.OvrdActLogAck := FALSE;
        END_IF
        
        IF FF.Ovrd.OvrdExpLogAck THEN
            
            pmpsTypeCode := 3;
            FormulateLogJson(FF);
            
            fbLogger(sMsg := 'Override released', eSevr:=TcEventSeverity.Warning);
            
            FF.Ovrd.OvrdExpLogAck := FALSE;
        END_IF
        
        IF FF.ClearAck THEN
            
            pmpsTypeCode := 8;
            FormulateLogJson(FF);
            
            fbLogger(sMsg := 'Fault cleared', eSevr:=TcEventSeverity.Info);
            
            FF.ClearAck := FALSE;
        END_IF
        
        
    END_IF
END_FOR

// Log registration fault cleared
tFFRegFail(CLK:=xFastFaultRegFail);
IF tFFRegFail.Q THEN
    fbJson.StartObject();
    fbJson.AddKey('pmps_typecode');
    fbJson.AddUdint(5);
    fbJson.AddKey('pmps_path');
    fbJson.AddString(sPath);
    fbJson.EndObject();
    fbJson.CopyDocument(pDoc:=fbLogger.sJson, SIZEOF(fbLogger.sJson));
    fbLogger(sMsg := 'Fast fault registration failure cleared. This may be bad as a fast fault could go unoticed.', 
        eSevr:=TcEventSeverity.Warning);  
END_IF

// Say hello
HelloTimer.IN := NOT HelloTimer.Q;
HelloTimer();
IF HelloTimer.IN THEN
    pmpsTypeCode := 10;
    FormulateLogJson(FF);   
    fbLogger(eSubsystem:=E_Subsystem.NILVALUE,
        eSevr := TcEventSeverity.Info,
        sMsg := 'FFO is alive');
    fbLogger.eSubsystem := E_Subsystem.MPS;
END_IF
END_METHOD

METHOD INTERNAL FormulateLogJson : STRING
VAR_INPUT
    FF : ST_FF;
END_VAR
fbJson.StartObject();
fbJson.AddKey('pmps_typecode');
fbJson.AddUdint(pmpsTypeCode);
fbJson.AddKey('pmps_path');
fbJson.AddString(FF.Info.sPath);
fbJson.AddKey('pmps_device_name');
fbJson.AddString(FF.Info.DevName);
fbJson.EndObject();
fbLogger.sJson := fbJson.GetDocument();
fbJson.ResetDocument();
END_METHOD

METHOD INTERNAL IdxCheckIn : BOOL
VAR_INPUT
    Idx : DINT;
    OK : BOOL;
    Reset : BOOL;
END_VAR
VAR
    stFF : ST_FF;
    BeamPermitted : BOOL;
END_VAR
Idx := LIMIT(1,Idx,FF_ARRAY_UPPER_BOUND);
stFF := THIS^.astFF[Idx];

// Updating internal fault state
stFF.OK := OK;

// Reset and latching logic
stFF.rtReset(CLK:=stFF.Reset (*epics*) OR Reset (*from other PLC logic *) );
stFF.Reset R= stFF.rtReset.Q;
stFF.bsFF(SET := stFF.rtReset.Q OR stFF.Info.AutoReset, RESET1:= NOT OK);    

BeamPermitted := stFF.bsFF.Q1 OR stFF.Ovrd.Active OR (i_xVeto AND stFF.Info.Vetoable);

// Fault generation    
IF NOT BeamPermitted THEN
    THIS^.xOK := FALSE; //Very clever, thanks Zach!
END_IF

// Fast fault accumulation
stFF.ftCountFault(CLK:=stFF.bsFF.Q1);
IF stFF.ftCountFault.Q THEN PMPS_GVL.AccumulatedFF := PMPS_GVL.AccumulatedFF + 1; END_IF

//Clear pushbuttons
stFF.Reset := FALSE;

// Log when this fault faults
stFF.FaultAck S= stFF.BeamPermitted AND NOT BeamPermitted;

// Log when this fault has cleared
stFF.ClearAck S= BeamPermitted AND NOT stFF.BeamPermitted;

stFF.BeamPermitted := BeamPermitted;

// Copy state back to ff struct
THIS^.astFF[Idx] := stFF;
END_METHOD

METHOD INTERNAL Register : BOOL
VAR_INPUT
    stFFInfo : ST_FFInfo := (
        sPath := '',
        Desc := '',
        TypeCode := 16#00,
        DevName := ''); // Fast fault information
        
END_VAR
VAR_OUTPUT
    FFOName : T_MaxString;
    Idx : UINT;
END_VAR
VAR
END_VAR
FFOName := THIS^.sPath;
Idx := THIS^.nIndex;

IF THIS^.nIndex <= FF_ARRAY_UPPER_BOUND THEN
    
    THIS^.astFF[MIN(THIS^.nIndex,FF_ARRAY_UPPER_BOUND)].Info:=stFFInfo;
    
    THIS^.nIndex := THIS^.nIndex + 1;
    
    Register := TRUE; // Add successful    
ELSE
    fbJson.StartObject();
    fbJson.AddKey('pmps_typecode');
    fbJson.AddUdint(4);
    fbJson.AddKey('pmps_path');
    fbJson.AddString(stFFInfo.sPath);
    fbJson.AddKey('pmps_device_name');
    fbJson.AddString(stFFInfo.DevName);
    fbJson.EndObject();
    fbLogger.sJson := fbJson.GetDocument();
    fbJson.ResetDocument();
    fbLogger(sMsg:='Fast fault registration failed. Too many fast faults on this FFO.',
        eSevr:=TcEventSeverity.Warning,
        eSubsystem:=E_Subsystem.MPS);
    xFastFaultRegFail := TRUE;
    Register := FALSE; // Failed to add name to list
END_IF
END_METHOD

END_FUNCTION_BLOCK

// MajorComponents/InterPlcComm/FB_ArbiterToSubSys_IO
(* Exchanges preemption requests and current beam state with subsystems in arbiter
network.

2019-12-2, A. Wallace

Use in conjunction with FB_SubSysToArbiter_IO.

This FB runs in the beamline arbiter PLC (BAP). There should be one of these for every
subsystem interfaced to the BAP. Each subsystem PLC should run a sibling FB_SubSysToArbiter_IO FB.

This FB and its sibling communicate through the ethercat connection between the subsystem PLC and the BAP.

*)
FUNCTION_BLOCK FB_ArbiterToSubSys_IO
VAR_INPUT
	RequestingSystemID	:	DWORD := PMPS_GVL.EXCLUDED_ASSERTION_ID; // System ID for making requests to the supreme arbiter
    sName : STRING := 'ArbiterToSubSys';
    Reset : BOOL;
END_VAR
VAR_OUTPUT
END_VAR
VAR_IN_OUT
	Arbiter	: FB_Arbiter;
    fbFFHWO : FB_HardwareFFOutput;
END_VAR
VAR
    
	i_RequestedBP AT %I*	:	ST_BeamParams_IO; // Requested BP from subsystem
    {attribute 'pytmc' := '
        pv: RequestedBP:FromSubSys
    '}
    RequestedBP: ST_BeamParams;
    
	o_CurrentBP AT %Q* : ST_BeamParams_IO; // Current BP set
    
    // EL6692 Diagnostics
    i_Connected AT %I* : BOOL; // SYNC Inputs^External device not connected !!! Doesn't really work.
    {attribute 'pytmc' := 'pv: WcState
        io: i
        field: DESC Working counter state.
        field: ZNAM OK
        field: ONAM Error'}
    i_WcState AT %I* : BOOL; // WcState^WcState
    {attribute 'pytmc' := 'pv: TxPDO_state
        io: i
        field: DESC PDO Transmission is OK
        field: ZNAM OK
        field: ONAM Error'}
    i_TxPDOState AT %I* : BOOL; // SYNC Inputs^TxPDO state
    {attribute 'pytmc' := 'pv: TxPDO_toggle
        io: i
        field: DESC PDO Transmission is OK
        field: ZNAM OK
        field: ONAM Error'}
    i_TxPDOToggle AT %I* : BOOL; // TxPDO toggle
    
    // Fast faults
    ffPMPSIO_Disconnect : FB_FastFault := (i_Desc:='Issue w/ arbiter interface to subsystem, verify subsystem is OK, or ethercat connection.'); // Fast fault for ethercat issues
    nActiveCohort : UDINT := 0; // Active cohort. Updated to the req. number from the sub system after request is confirmed.
    nRequestedCohort : UDINT := 0;
    rtToggle : R_TRIG;

	
END_VAR


// Incoming request from subsystem PLC
RequestedBP := IO_TO_BP(i_RequestedBP);

// Update Arbiter with our request
rtToggle(CLK:= i_RequestedBP.xValid); // If interface resumes, reset/catch up
// xValid will go false if the PLC program on the other side is stopped. Ironically the ethercat interface continues happily.
// If subsystem cohort has incremented, update beam parameter request with our arbiter
IF i_RequestedBP.nCohortInt > nRequestedCohort OR rtToggle.Q THEN 
    Arbiter.RemoveRequest(RequestingSystemID);
    Arbiter.AddRequest(RequestingSystemID, RequestedBP);
    nRequestedCohort := i_RequestedBP.nCohortInt;
END_IF


// Check if latest request is acknowledged by this arbiter
// Acknowledgement happens after an arbitration cycle, which means if RequestedCohort just incremented
// due to a new request, CheckRequest will be false.
IF Arbiter.CheckRequest(RequestingSystemID) THEN
    nActiveCohort := nRequestedCohort; // If it is, then the active cohort is set to the requested cohort number.
END_IF

// Sending current beam parameter set to subsystems 
o_CurrentBP := BP_TO_IO(PMPS_GVL.stCurrentBeamParameters);
o_CurrentBP.nCohortInt := nActiveCohort;


//////////////////////////////////////
// Verifying the ethercat interface health
/////////////////////////////////////
// Both of these values should be 0 for a fully valid exchange
ffPMPSIO_Disconnect.i_xOK := NOT i_WcState AND NOT i_TxPDOState;

ffPMPSIO_Disconnect(
    io_fbFFHWO := fbFFHWO,
    i_xReset := Reset,
    i_DevName := sName,
    i_TypeCode:=5);

END_FUNCTION_BLOCK

// MajorComponents/InterPlcComm/FB_SubSysToArbiter_IO
// Use on a subsystem PLC to request from the arbiter
// Run at the top of your cycle to receive the latest BP
FUNCTION_BLOCK FB_SubSysToArbiter_IO IMPLEMENTS I_HigherAuthority
VAR_INPUT
    Reset : BOOL; // Fast fault reset
    sName : STRING := 'SubSysToArbiter';
END_VAR
VAR_OUTPUT
END_VAR
VAR_IN_OUT
	Arbiter	: FB_Arbiter;
    fbFFHWO : FB_HardwareFFOutput;
END_VAR
VAR
    {attribute 'TcLinkTo' := 'TIIB[PMPS_PRE]^IO Inputs^CurrentBP'}
    i_stCurrentBP    AT %I* :    ST_BeamParams_IO;
    {attribute 'TcLinkTo' := 'TIIB[PMPS_PRE]^IO Outputs^RequestedBP'}
    q_stRequestedBP AT %Q* :    ST_BeamParams_IO;
    {attribute 'pytmc' := 'pv: TxPDO_toggle
        io: i'}
    {attribute 'TcLinkTo' := 'TIIB[PMPS_PRE]^SYNC Inputs^TxPDO toggle'}
    xTxPDO_toggle    AT     %I* :    BIT;
    {attribute 'pytmc' := 'pv: TxPDO_state
        io: i'}
    {attribute 'TcLinkTo' := 'TIIB[PMPS_PRE]^SYNC Inputs^TxPDO state'}
    xTxPDO_state    AT    %I*    :    BIT;
    
    
    // Fast faults
    ffPMPSIO_Disconnect : FB_FastFault := (i_Desc:='Arbiter network interface disconnected or not OP',i_DevName := sName);
    
    // A request is not considered included until the active cohort number is >= the request cohort number.
    {attribute 'pytmc' := 'pv: RequestCohort
        io: i'}
    nRequestCohort : UDINT := 0; // Request cohort
    {attribute 'pytmc' := 'pv: ActiveCohort
        io: i'}
    nActiveCohort : UDINT := 0; // Active cohort, updated by incoming BP from arbiter PLC, in the ElevateRequest arbiter call

END_VAR

//Receiving current BP state
PMPS_GVL.stCurrentBeamParameters := IO_TO_BP(i_stCurrentBP);
PMPS_GVL.stCurrentBeamParameters.xValidToggle := xTxPDO_toggle; // This line must follow the one above. Sequence is important.

// Forwarding BP request for the subsystem
Arbiter.ElevateRequest(THIS^);

//Broadcasting current request
PMPS_GVL.stRequestedBeamParameters := IO_TO_BP(q_stRequestedBP);


q_stRequestedBP.xValid := TRUE; // This is set and held true here every cycle to prove the PLC on this side is still running

ffPMPSIO_Disconnect(
    i_xOK := xTxPDO_state = 0,
    io_fbFFHWO := fbFFHWO,
    i_xReset := Reset,
    i_DevName := sName,
    i_TypeCode := 6,
    i_xVetoable := FALSE
    );

METHOD CheckRequest : BOOL
VAR_INPUT
	nReqID	: DWORD;
END_VAR
VAR_INST
    xFirstTime : BOOL := TRUE;
    nId : DWORD;
END_VAR
// Check this id matches what we've seen before
IF xFirstTime THEN
    nId := nReqId;
ELSIF nId <> nReqId THEN
    PMPS_GVL.fbLog(sMsg := 'SubSysToArbiter Check mismatched with a different ID', eSevr := TcEventSeverity.Error);
    RETURN;
END_IF

nActiveCohort := ULINT_TO_UDINT(i_stCurrentBP.nCohortInt);

// i_stCurrentBP.nCohortInt is incremented by the FB_ArbiterToSubSys block on the other side of the EL669* interface
CheckRequest := nRequestCohort <= nActiveCohort;
END_METHOD

METHOD RequestBP : BOOL
VAR_INPUT
	(*StateID of state requesting beam parameter set*)
	nReqID	: DWORD;
	(*Requested beam params*)
	stReqBP	: ST_BeamParams;
END_VAR
// Check the request is coming from the same source we're used to

// Update internal BP request struct
q_stRequestedBP := BP_TO_IO(stReqBP);

nRequestCohort := nRequestCohort + 1;

// Mark the current cohort id
q_stRequestedBP.nCohortInt := nRequestCohort;

RequestBP := TRUE;
END_METHOD

END_FUNCTION_BLOCK

// MajorComponents/PhotonEnergyInterface/F_CalculatePhotonEnergy
FUNCTION F_CalculatePhotonEnergy : LREAL
VAR_INPUT
    (* Electron energy in GeV *)
    fElectronEnergy_GeV : LREAL;
    (* Undulator period in mm *)
    fUndulatorPeriod_mm : LREAL;
    (* Unitless undulator K parameter / strength *)
    fUndulatorStrength : LREAL;
END_VAR

VAR
    fDenominator: LREAL;
END_VAR

VAR CONSTANT
    (* GeV [electron rest mass/energy] *)
    m_e : LREAL := 0.0005109989461;
    (* Js [Planck's constant] *)
    h 	: LREAL := 6.62607004E-34;
    (* C [electron charge] *)
    e 	: LREAL := 1.6021766208E-19;
    (* m/s, speed of light *)
    c 	: LREAL := 299792458;

END_VAR

(*

Reference Python implementation

def calculate_photon_energy(electron_energy, period, k):
    '''
    Calculate photon energy, in eV.

    Parameters
    ----------
    electron_energy : float
        Electron energy in GeV

    period : float
        Undulator period, in mm

    k : float
        Undulator K parameter (strength), unitless
    '''
    m_e = 0.0005109989461  # GeV [electron rest mass/energy]
    h = 6.62607004e-34  # Js [Planck's constant]
    e = 1.6021766208e-19  # C [electron charge]
    c = 299792458  # m/s, speed of light
    return ((2. * (electron_energy / m_e) ** 2 * h * c) /
            (e * period * 1e-3 * (1 + k ** 2 / 2.)))

*)
fDenominator := (e * fUndulatorPeriod_mm * 1E-3 * (1.0 + EXPT(fUndulatorStrength, 2.0) / 2.0));
F_CalculatePhotonEnergy := (2.0 * EXPT(fElectronEnergy_GeV / m_e, 2.0) * h * c) / MAX(fDenominator, 4.94065645841247E-324);

END_FUNCTION

// MajorComponents/PhotonEnergyInterface/FB_AcceleratorLinks
FUNCTION_BLOCK FB_AcceleratorLinks
VAR_INPUT

END_VAR

VAR_OUTPUT
END_VAR


VAR

    {attribute 'pytmc' := '
        pv: eEnrg:Hgvpu
        link: BEND:DMPH:400:BACT
        field: EGU GeV
    '}
    fbHgvpuElectronEnergy : FB_LREALFromEPICS;

    {attribute 'pytmc' := '
        pv: eEnrg:SXU
        link: BEND:DMPS:400:BACT
        field: EGU GeV
    '}
    fbSxuElectronEnergy : FB_LREALFromEPICS;

END_VAR

fbHgvpuElectronEnergy();
fbSxuElectronEnergy();

END_FUNCTION_BLOCK

// MajorComponents/PhotonEnergyInterface/FB_Hgvpu
FUNCTION_BLOCK FB_Hgvpu
VAR_INPUT
    fbElectronEnergy : REFERENCE TO FB_LREALFromEPICS;
END_VAR

VAR_OUTPUT
	{attribute 'pytmc' := '
        pv: CurrentPhotonEnergy
		io: i
        field: DESC Calculated current photon energy
        field: PREC 3
        field: EGU eV
    '}
	fCurrentPhotonEnergy : LREAL;
	{attribute 'pytmc' := '
        pv: TargetPhotonEnergy
		io: i
        field: DESC Calculated desired photon energy
        field: PREC 3
        field: EGU eV
    '}
	fTargetPhotonEnergy : LREAL;
	    {attribute 'pytmc' := '
        pv: SeedUndulatorNumber
		io: i
        field: DESC Seed undulator number
    '}
	nSeedUndulator : UDINT; // Set to zero when no undulators are active
END_VAR


VAR
    // From lcls-srv01: grep -e KDes  /u1/lcls/epics/ioc/data/ioc-undh-uc*/iocInfo/IOC.pvlist |sort

    {attribute 'pytmc' := 'pv: 24; link: 2450:'}
    fbSegment_24 : FB_UndulatorSegment;

    {attribute 'pytmc' := 'pv: 25; link: 2550:'}
    fbSegment_25 : FB_UndulatorSegment;

    {attribute 'pytmc' := 'pv: 26; link: 2650:'}
    fbSegment_26 : FB_UndulatorSegment;

    {attribute 'pytmc' := 'pv: 27; link: 2750:'}
    fbSegment_27 : FB_UndulatorSegment;

    {attribute 'pytmc' := 'pv: 29; link: 2950:'}
    fbSegment_29 : FB_UndulatorSegment;

    {attribute 'pytmc' := 'pv: 30; link: 3050:'}
    fbSegment_30 : FB_UndulatorSegment;

    {attribute 'pytmc' := 'pv: 31; link: 3150:'}
    fbSegment_31 : FB_UndulatorSegment;

    {attribute 'pytmc' := 'pv: 32; link: 3250:'}
    fbSegment_32 : FB_UndulatorSegment;

    {attribute 'pytmc' := 'pv: 33; link: 3350:'}
    fbSegment_33 : FB_UndulatorSegment;

    {attribute 'pytmc' := 'pv: 34; link: 3450:'}
    fbSegment_34 : FB_UndulatorSegment;

    {attribute 'pytmc' := 'pv: 35; link: 3550:'}
    fbSegment_35 : FB_UndulatorSegment;

    {attribute 'pytmc' := 'pv: 36; link: 3650:'}
    fbSegment_36 : FB_UndulatorSegment;

    {attribute 'pytmc' := 'pv: 37; link: 3750:'}
    fbSegment_37 : FB_UndulatorSegment;

    {attribute 'pytmc' := 'pv: 38; link: 3850:'}
    fbSegment_38 : FB_UndulatorSegment;

    {attribute 'pytmc' := 'pv: 39; link: 3950:'}
    fbSegment_39 : FB_UndulatorSegment;

    {attribute 'pytmc' := 'pv: 40; link: 4050:'}
    fbSegment_40 : FB_UndulatorSegment;

    {attribute 'pytmc' := 'pv: 41; link: 4150:'}
    fbSegment_41 : FB_UndulatorSegment;

    {attribute 'pytmc' := 'pv: 42; link: 4250:'}
    fbSegment_42 : FB_UndulatorSegment;

    {attribute 'pytmc' := 'pv: 43; link: 4350:'}
    fbSegment_43 : FB_UndulatorSegment;

    {attribute 'pytmc' := 'pv: 44; link: 4450:'}
    fbSegment_44 : FB_UndulatorSegment;

    {attribute 'pytmc' := 'pv: 45; link: 4550:'}
    fbSegment_45 : FB_UndulatorSegment;

    {attribute 'pytmc' := 'pv: 46; link: 4650:'}
    fbSegment_46 : FB_UndulatorSegment;

    fbSegment : ARRAY [PMPS_GVL.iLowBound_LUnd..PMPS_GVL.iHighBound_LUnd] OF POINTER TO FB_UndulatorSegment;
    fbCurrentSegment : REFERENCE TO FB_UndulatorSegment;

    iIndex : UDINT;

    bInitialized : BOOL := FALSE;

END_VAR

VAR CONSTANT

END_VAR

IF NOT bInitialized THEN
	Init();
END_IF

UndAdrUpdate();

nSeedUndulator := 0;

FOR iIndex := PMPS_GVL.iLowBound_LUnd TO PMPS_GVL.iHighBound_LUnd DO
    IF fbSegment[iIndex] <> 0 THEN
        fbCurrentSegment REF= fbSegment[iIndex]^;
        fbCurrentSegment(fbElectronEnergy:=fbElectronEnergy);
		
		//Mark the seed undulator, first undulator operating within K bounds
		IF fbCurrentSegment.xActive AND nSeedUndulator = 0 THEN
			nSeedUndulator := iIndex;
			fCurrentPhotonEnergy := fbCurrentSegment.fPhotonEnergyAct;
			fTargetPhotonEnergy := fbCurrentSegment.fPhotonEnergyDes;
		END_IF
    END_IF
END_FOR

IF nSeedUndulator = 0 THEN
	fCurrentPhotonEnergy := 0;
	fTargetPhotonEnergy := 0;
END_IF

ACTION Init:

UndAdrUpdate();


    FOR iIndex := PMPS_GVL.iLowBound_LUnd TO PMPS_GVL.iHighBound_LUnd DO
            IF fbSegment[iIndex] <> 0 THEN
            fbCurrentSegment REF= fbSegment[iIndex]^;
            fbCurrentSegment.fPeriod_mm := PMPS_GVL.fPeriod_mm_LUnd;
			fbCurrentSegment.fLowK := PMPS_GVL.fLowK_LUnd;
			fbCurrentSegment.fHiK := PMPS_GVL.fHiK_LUnd;
        END_IF
    END_FOR

    bInitialized := TRUE;
END_ACTION

ACTION UndAdrUpdate:
    fbSegment[24] := ADR(fbSegment_24);
    fbSegment[25] := ADR(fbSegment_25);
    fbSegment[26] := ADR(fbSegment_26);
    fbSegment[27] := ADR(fbSegment_27);
    fbSegment[28] := 0;
    fbSegment[29] := ADR(fbSegment_29);
    fbSegment[30] := ADR(fbSegment_30);
    fbSegment[31] := ADR(fbSegment_31);
    fbSegment[32] := ADR(fbSegment_32);
    fbSegment[33] := ADR(fbSegment_33);
    fbSegment[34] := ADR(fbSegment_34);
    fbSegment[35] := ADR(fbSegment_35);
    fbSegment[36] := ADR(fbSegment_36);
    fbSegment[37] := ADR(fbSegment_37);
    fbSegment[38] := ADR(fbSegment_38);
    fbSegment[39] := ADR(fbSegment_39);
    fbSegment[40] := ADR(fbSegment_40);
    fbSegment[41] := ADR(fbSegment_41);
    fbSegment[42] := ADR(fbSegment_42);
    fbSegment[43] := ADR(fbSegment_43);
    fbSegment[44] := ADR(fbSegment_44);
    fbSegment[45] := ADR(fbSegment_45);
    fbSegment[46] := ADR(fbSegment_46);
END_ACTION

END_FUNCTION_BLOCK

// MajorComponents/PhotonEnergyInterface/FB_UndulatorSegment
FUNCTION_BLOCK FB_UndulatorSegment
VAR_INPUT
    (* Undulator period in millimeters, to be set by subclasses *)
    fPeriod_mm : LREAL := 1.0;
    fbElectronEnergy : REFERENCE TO FB_LREALFromEPICS;
	
	fLowK : LREAL := 0;
	fHiK : LREAL := 6;
	fKRangeHyst : LREAL := 0.01;
END_VAR

VAR_OUTPUT
    {attribute 'pytmc' := '
        pv: eVAct
        field: DESC Calculated photon energy
        field: PREC 3
        field: EGU eV
    '}
    fPhotonEnergyAct : LREAL;

    {attribute 'pytmc' := '
        pv: eVDes
        field: DESC Calculated desired photon energy
        field: PREC 3
        field: EGU eV
    '}
    fPhotonEnergyDes : LREAL;
	
	{attribute 'pytmc' := '
        pv: Active
		io: i
        field: DESC Undulator is considered active
    '}
	xActive : BOOL; // Undulator is considered active
END_VAR

VAR
    {attribute 'pytmc' := '
        pv: KDes
        link: KDes
    '}
    fbKDesired : FB_LREALFromEPICS;

    {attribute 'pytmc' := '
        pv: KAct
        link: KAct
    '}
    fbKActual : FB_LREALFromEPICS;

END_VAR

fbKDesired();
fbKActual();

IF __ISVALIDREF(fbElectronEnergy) THEN

    IF fbKActual.bValid AND fbElectronEnergy.bValid THEN
        fPhotonEnergyAct := F_CalculatePhotonEnergy(
            fElectronEnergy_GeV:=fbElectronEnergy.fValue,
            fUndulatorPeriod_mm:=fPeriod_mm,
            fUndulatorStrength:=fbKActual.fValue
        );
		
		//Set this undulator active if actual K is within operational range
		xActive S= fLowK <= fbKActual.fValue AND fbKActual.fValue <= fHiK AND
		(fbKActual.bValid AND fbKActual.bValid);
		xActive R= (fLowK - fKRangeHyst) > fbKActual.fValue OR fbKActual.fValue > (fHiK + fKRangeHyst) OR
					(NOT fbKActual.bValid OR NOT fbKActual.bValid);
    END_IF

    IF fbKDesired.bValid AND fbElectronEnergy.bValid THEN
        fPhotonEnergyDes := F_CalculatePhotonEnergy(
            fElectronEnergy_GeV:=fbElectronEnergy.fValue,
            fUndulatorPeriod_mm:=fPeriod_mm,
            fUndulatorStrength:=fbKDesired.fValue
        );
    END_IF

END_IF

END_FUNCTION_BLOCK

// MajorComponents/PhotonEnergyInterface/FB_LPhotonEnergy
FUNCTION_BLOCK FB_LPhotonEnergy
VAR_INPUT
END_VAR
VAR_OUTPUT
END_VAR
VAR_IN_OUT
	BP : ST_BeamParams;
END_VAR
VAR
	{attribute 'pytmc' := '
        pv: eEnrg
        link: BEND:DMPH:400:BACT
        field: EGU GeV
    '}
    fbHgvpuElectronEnergy : FB_LREALFromEPICS;
	
	{attribute 'pytmc' := '
        pv: UND
        link: USEG:UNDH:
    '}
    fbHgvpu : FB_Hgvpu;
	
	nCurrentPhotonEnergyBitmask : UINT;
	nTargetPhotonEnergyBitmask : UINT;
END_VAR

// Update PVs
fbHgvpuElectronEnergy();

fbHgvpu(fbElectronEnergy:=fbHgvpuElectronEnergy);

//Update BP
nCurrentPhotonEnergyBitmask := F_eVRangeCalculator(fbHgvpu.fCurrentPhotonEnergy, nCurrentPhotonEnergyBitmask);
nTargetPhotonEnergyBitmask := F_eVRangeCalculator(fbHgvpu.fTargetPhotonEnergy, nTargetPhotonEnergyBitmask);

BP.neVRange := nCurrentPhotonEnergyBitmask OR nTargetPhotonEnergyBitmask;

END_FUNCTION_BLOCK

// MajorComponents/PhotonEnergyInterface/FB_SXU
FUNCTION_BLOCK FB_SXU
VAR_INPUT
    fbElectronEnergy : REFERENCE TO FB_LREALFromEPICS;
END_VAR

VAR_OUTPUT
END_VAR



VAR
    // From lcls-srv01: grep -e KDes  /u1/lcls/epics/ioc/data/sioc-unds-uc*/iocInfo/IOC.pvlist |sort


    {attribute 'pytmc' := 'pv: 26; link: 2650:'}
    fbSegment_26 : FB_UndulatorSegment;

    {attribute 'pytmc' := 'pv: 27; link: 2750:'}
    fbSegment_27 : FB_UndulatorSegment;

    {attribute 'pytmc' := 'pv: 28; link: 2850:'}
    fbSegment_28 : FB_UndulatorSegment;

    {attribute 'pytmc' := 'pv: 29; link: 2950:'}
    fbSegment_29 : FB_UndulatorSegment;

    {attribute 'pytmc' := 'pv: 30; link: 3050:'}
    fbSegment_30 : FB_UndulatorSegment;

    {attribute 'pytmc' := 'pv: 31; link: 3150:'}
    fbSegment_31 : FB_UndulatorSegment;

    {attribute 'pytmc' := 'pv: 32; link: 3250:'}
    fbSegment_32 : FB_UndulatorSegment;

    {attribute 'pytmc' := 'pv: 33; link: 3350:'}
    fbSegment_33 : FB_UndulatorSegment;

    {attribute 'pytmc' := 'pv: 34; link: 3450:'}
    fbSegment_34 : FB_UndulatorSegment;

    {attribute 'pytmc' := 'pv: 36; link: 3650:'}
    fbSegment_36 : FB_UndulatorSegment;

    {attribute 'pytmc' := 'pv: 37; link: 3750:'}
    fbSegment_37 : FB_UndulatorSegment;

    {attribute 'pytmc' := 'pv: 38; link: 3850:'}
    fbSegment_38 : FB_UndulatorSegment;

    {attribute 'pytmc' := 'pv: 39; link: 3950:'}
    fbSegment_39 : FB_UndulatorSegment;

    {attribute 'pytmc' := 'pv: 40; link: 4050:'}
    fbSegment_40 : FB_UndulatorSegment;

    {attribute 'pytmc' := 'pv: 41; link: 4150:'}
    fbSegment_41 : FB_UndulatorSegment;

    {attribute 'pytmc' := 'pv: 42; link: 4250:'}
    fbSegment_42 : FB_UndulatorSegment;

    {attribute 'pytmc' := 'pv: 43; link: 4350:'}
    fbSegment_43 : FB_UndulatorSegment;

    {attribute 'pytmc' := 'pv: 44; link: 4450:'}
    fbSegment_44 : FB_UndulatorSegment;

    {attribute 'pytmc' := 'pv: 45; link: 4550:'}
    fbSegment_45 : FB_UndulatorSegment;

    {attribute 'pytmc' := 'pv: 46; link: 4650:'}
    fbSegment_46 : FB_UndulatorSegment;

    {attribute 'pytmc' := 'pv: 47; link: 4750:'}
    fbSegment_47 : FB_UndulatorSegment;



    fbSegment : ARRAY [iLowBound..iHighBound] OF POINTER TO FB_UndulatorSegment;
    fbCurrentSegment : REFERENCE TO FB_UndulatorSegment;

    iIndex : UDINT;

    bInitialized : BOOL := FALSE;

END_VAR

VAR CONSTANT
    {attribute 'pytmc' := 'pv: FirstSegment; io: i'}
    iLowBound  : UDINT := 26;
    {attribute 'pytmc' := 'pv: LastSegment; io: i'}
    iHighBound : UDINT := 47;
    {attribute 'pytmc' := '
        pv: Period
        io: i
        field: EGU mm
    '}
    fPeriod_mm : LREAL := 39.0;
END_VAR



IF NOT bInitialized THEN

    fbSegment[26] := ADR(fbSegment_26);
    fbSegment[27] := ADR(fbSegment_27);
    fbSegment[28] := ADR(fbSegment_28);
    fbSegment[29] := ADR(fbSegment_29);
    fbSegment[30] := ADR(fbSegment_30);
    fbSegment[31] := ADR(fbSegment_31);
    fbSegment[32] := ADR(fbSegment_32);
    fbSegment[33] := ADR(fbSegment_33);
    fbSegment[34] := ADR(fbSegment_34);
    fbSegment[35] := 0;
    fbSegment[36] := ADR(fbSegment_36);
    fbSegment[37] := ADR(fbSegment_37);
    fbSegment[38] := ADR(fbSegment_38);
    fbSegment[39] := ADR(fbSegment_39);
    fbSegment[40] := ADR(fbSegment_40);
    fbSegment[41] := ADR(fbSegment_41);
    fbSegment[42] := ADR(fbSegment_42);
    fbSegment[43] := ADR(fbSegment_43);
    fbSegment[44] := ADR(fbSegment_44);
    fbSegment[45] := ADR(fbSegment_45);
    fbSegment[46] := ADR(fbSegment_46);
    fbSegment[47] := ADR(fbSegment_47);

    FOR iIndex := iLowBound TO iHighBound DO
            IF fbSegment[iIndex] <> 0 THEN
            fbCurrentSegment REF= fbSegment[iIndex]^;
            fbCurrentSegment.fPeriod_mm := fPeriod_mm;
        END_IF
    END_FOR
    bInitialized := TRUE;
END_IF

FOR iIndex := iLowBound TO iHighBound DO
    IF fbSegment[iIndex] <> 0 THEN
        fbCurrentSegment REF= fbSegment[iIndex]^;
        fbCurrentSegment(fbElectronEnergy:=fbElectronEnergy);
    END_IF
END_FOR

END_FUNCTION_BLOCK

// MajorComponents/PMPS_MPS_Interface/FB_BeamClassOutputs
(*
Sets the beam class assertion lines for a given beam class.
*)
FUNCTION_BLOCK FB_BeamClassOutputs
VAR_INPUT
    BP : ST_BeamParams;
END_VAR
VAR_OUTPUT
END_VAR
VAR
    nBeamClass   :    BYTE;
    wBeamClass    :    BYTE;

    InitCounter: BYTE;
    counter    :    INT;
    
    // Beam class lines are restricted to 8 channels in the current design, since
    // there are no plans to use all 16. Channels 1-7 may be allocated to any other
    // beam classes so long as they are ordered least to greatest.
    // Channel 8 is reserved for full beam.
    {attribute 'pytmc' := 'pv: BeamClassChannel
        io: i
        field: DESC Hardwire channel state'}
        epicsBitmap : WORD;
        
    {attribute 'TcLinkTo' := '[1] := TIIB[PMPS_Premp]^Channel 1^Output;
                              [2] := TIIB[PMPS_Premp]^Channel 2^Output;
                              [3] := TIIB[PMPS_Premp]^Channel 3^Output;
                              [4] := TIIB[PMPS_Premp]^Channel 4^Output;
                              
                              [5] := TIIB[PMPS_Premp]^Channel 5^Output;
                              [6] := TIIB[PMPS_Premp]^Channel 6^Output;
                              [7] := TIIB[PMPS_Premp]^Channel 7^Output;
                              [8] := TIIB[PMPS_Premp]^Channel 8^Output;'} // 8 - Full beam
    q_BC_ASSERTION_LINES    AT    %Q*    : ARRAY [1..MAX_BEAM_CLASS_LINES] OF    BOOL;
END_VAR
VAR CONSTANT
    MAX_BEAM_CLASS_LINES : BYTE := 8;
    BC_1HZ : BYTE := 1;
    BC_10HZ : BYTE := 2;
    BC_FULL : BYTE := 16;
END_VAR


// Determine BC
IF BP.nRate >= 120 THEN
    nBeamClass := BC_FULL;
ELSIF BP.nRate >= 10 THEN
    nBeamClass := BC_10HZ;
ELSIF BP.nRate >= 1 THEN
    nBeamClass := BC_1HZ;
ELSE
	nBeamClass := 0;
END_IF


//Assert Beam Class
////////////////////////////////////
//0x0 = 0000 0000 0000 0000
//0x1 = 0000 0000 0000 0001
//0xF = 1111 1111 1111 1111

//Initialize BC lines to zero on every pass
FOR InitCounter := 1 TO MAX_BEAM_CLASS_LINES DO
    q_BC_ASSERTION_LINES[InitCounter] := FALSE;
END_FOR

//Set BC lines according to beam class
//A BC of 0x0 would pass over this loop, setting none of the lines high
// , as FOR loops check the initialized variable at the top to see if it's >
// than the "TO" variable.
FOR wBeamClass:=1 TO MIN(MAX_BEAM_CLASS_LINES-1, nBeamClass) DO
    q_BC_ASSERTION_LINES[wBeamClass] := TRUE;
END_FOR

q_BC_ASSERTION_LINES[8] := nBeamClass = 16; //Set channel 8 true if BC is 16


// Readbacks for EPICS
epicsBitmap.0 := q_BC_ASSERTION_LINES[1];
epicsBitmap.1 := q_BC_ASSERTION_LINES[2];
epicsBitmap.2 := q_BC_ASSERTION_LINES[3];
epicsBitmap.3 := q_BC_ASSERTION_LINES[4];

epicsBitmap.4 := q_BC_ASSERTION_LINES[5];
epicsBitmap.5 := q_BC_ASSERTION_LINES[6];
epicsBitmap.6 := q_BC_ASSERTION_LINES[7];
epicsBitmap.7 := q_BC_ASSERTION_LINES[8];

END_FUNCTION_BLOCK

// MajorComponents/PMPS_MPS_Interface/FB_CTLS_Outputs
(*
Controls auxiliary beam class outputs.

1-3 are mapped to control the Cu beamline rate via the LCLS II MPS.

Maps beam rate requests to 1, 10, or full rate beam for Cu linac.

*)
FUNCTION_BLOCK FB_CTLS_Outputs
VAR_INPUT
    BP    :    ST_BeamParams;
END_VAR
VAR_OUTPUT
END_VAR
VAR
    {attribute 'pytmc' := 'pv: CTLSChannel
        io: i
        field: DESC CTLS Rate Control hardwire channel state'}
    epicsBitmap : WORD;
        
    {attribute 'TcLinkTo' := '[1] := TIIB[PMPS_Premp]^Channel 9^Output;
                              [2] := TIIB[PMPS_Premp]^Channel 10^Output;
                              [3] := TIIB[PMPS_Premp]^Channel 11^Output;'}
    q_CLTS_ASSERTION_LINES    AT    %Q*    : ARRAY [1..3] OF    BOOL;  
    
    
    
END_VAR


// CLTS 1Hz
q_CLTS_ASSERTION_LINES[1] := BP.nRate >= 1;
// CLTS 10Hz
q_CLTS_ASSERTION_LINES[2] := BP.nRate >= 10;
// CLTS Full rate
q_CLTS_ASSERTION_LINES[3] := BP.nRate >= 120;


epicsBitMap.0 := q_CLTS_ASSERTION_LINES[1];
epicsBitMap.1 := q_CLTS_ASSERTION_LINES[2];
epicsBitMap.2 := q_CLTS_ASSERTION_LINES[3];

END_FUNCTION_BLOCK

// MajorComponents/PMPS_MPS_Interface/FB_PhotonEnergyWatcher
(*
A. Wallace 2019-4-22
The photon energy watcher ensures the current and target photon energy is within
the arbirated bounds. Target in this case means, the calculated target photon energy
from the PVs that control the mechatronics of the undulators/ the electron energy.

If there are control PVs that match the monitor PVs, the control PVs are used to 
calculate a "target" photon energy. This is supposed to cover when the undulators/
electron energy is transitioning.

The abritrated bounds come from a simple AND of all the permitted ranges. See
the arbitrate action of the arbiter FB.

Note, this protection logic does not account for beam-off when determining fast-fault
status. If a device is requesting a limited range of eV, this request must be honored,
regardless of current beam-rate.
*)
FUNCTION_BLOCK FB_PhotonEnergyWatcher
VAR_INPUT
    i_stCurrentBeamParams    :    ST_BeamParams; //Link to global beam params
    i_stMachineTargetBeamParams    :    ST_BeamParams; //Link to global machine target beam params
    i_stRequestedBeamParams    :    ST_BeamParams; //Link to arbiter output or beam param. requestor
    // Reset fault
    i_xReset: BOOL;
    sName : STRING := 'PhotonEnergyWatcher';
END_VAR
VAR_OUTPUT
END_VAR
VAR_IN_OUT
    io_fbFFHWO    :    FB_HardwareFFOutput;
END_VAR
VAR
    xPhotonEnergyWithinBounds    :    BOOL;
    fbFF    :    FB_FastFault :=(
        i_DevName := sName,
        i_Desc := 'Fault occurs when the calculated machine photon energy (K value calculated by undulator gap, and electron energy) falls outside the permitted range.',
        i_TypeCode := 7 );
        
   {attribute 'pytmc' := '
        pv: ResidualPhotonEnergies
		io: i
        archive: 1Hz monitor
        field: DESC Portions of beam eV not permitted
        field: EGU eV-bitmask
    '}
    evResidual : WORD;
END_VAR

xPhotonEnergyWithinBounds := (i_stCurrentBeamParams.neVRange AND i_stRequestedBeamParams.neVRange) = i_stCurrentBeamParams.neVRange;

evResidual := (i_stCurrentBeamParams.neVRange XOR i_stRequestedBeamParams.neVRange) AND i_stCurrentBeamParams.neVRange;

fbFF(i_xOK := xPhotonEnergyWithinBounds,
    i_xReset := i_xReset,
    io_fbFFHWO := io_fbFFHWO);

END_FUNCTION_BLOCK

// MajorComponents/SimulationFB/FB_eVSimulator
(* eV Simulator
A. Wallace 2019-8-30

Adds noise to the eV and changes eV position occasionally.
*)
FUNCTION_BLOCK FB_eVSimulator
VAR_INPUT
    NoiseLevel	:	REAL	:= 0; // eV Noise
    ChangeTime : TIME := T#10S;
END_VAR
VAR_OUTPUT
    eV	:	REAL := 300;
END_VAR
VAR
    eVRange : REAL := 1600;
    timer: TON;
    eVRand	:	DRAND :=(Seed:=0);
    NoiseRand : DRAND := (Seed:=0);
END_VAR


timer(in:=TRUE, PT:=ChangeTime);

//Occasionally change eV
IF timer.Q THEN
    timer(in:=FALSE);
    eVRand();
    eV := LIMIT(0, eVRange*LREAL_TO_REAL(eVRand.Num), eVRange);
END_IF

// Noise generation
NoiseRand();
eV := eV + NoiseLevel*LREAL_TO_REAL(NoiseRand.Num);
NoiseRand();
eV := LIMIT(0, ev - NoiseLevel*LREAL_TO_REAL(NoiseRand.Num), eVRange);

END_FUNCTION_BLOCK

// MajorComponents/SimulationFB/FB_MachineSimulator
(* Simulates the machine responding to requests by adding a bit of delay/ ramps
*)
FUNCTION_BLOCK FB_MachineSimulator
VAR_INPUT
    i_stAssertedParams    :    ST_BeamParams;
    i_xFault    :    BOOL;
    
    xEnableAtt : BOOL;
    xEnablePE : BOOL;
    xEnableRate : BOOL;
END_VAR
VAR_IN_OUT
    iq_stMachineParams    :    ST_BeamParams;
END_VAR
VAR
    nTargetTran: UINT;
    tonTranTimer    :    TON := (
        PT := T#2S
        );
    fTargetPP_mJ: REAL;
    tonPPETimer: TON := (
        PT := T#2S
    );
END_VAR


//Attenuation
IF xEnableAtt THEN
    IF i_stAssertedParams.nTran <> nTargetTran THEN
        tonTranTimer(IN:=FALSE);
        nTargetTran := i_stAssertedParams.nTran;
    ELSIF NOT tonTranTimer.Q THEN
        tonTranTimer(IN:=TRUE);
    ELSE
        iq_stMachineParams.nTran := nTargetTran;
    END_IF
END_IF
    
//Pulse Energy
IF xEnablePE THEN
    IF i_stAssertedParams.fPP_mJ <> fTargetPP_mJ THEN
        tonPPETimer(IN:=FALSE);
        fTargetPP_mJ := i_stAssertedParams.fPP_mJ;
    ELSIF NOT tonTranTimer.Q THEN
        tonPPETimer(IN:=TRUE);
    ELSE
        iq_stMachineParams.fPP_mJ := fTargetPP_mJ;
    END_IF
END_IF

//Rate
IF xEnableRate THEN
    IF i_xFault THEN
        iq_stMachineParams.nRate := 0;
    ELSE
        iq_stMachineParams.nRate := i_stAssertedParams.nRate;
    END_IF
END_IF

END_FUNCTION_BLOCK

// MajorComponents/Stoppers/FB_KStopper
FUNCTION_BLOCK FB_KStopper EXTENDS FB_StopperWatcher
VAR_INPUT
END_VAR
VAR_OUTPUT
END_VAR
VAR_IN_OUT
END_VAR
VAR
END_VAR

SUPER^(stCurrentBP:=SUPER^.stCurrentBP);

METHOD FB_init : BOOL
VAR_INPUT
    bInitRetains : BOOL; // if TRUE, the retain variables are initialized (warm start / cold start)
    bInCopyCode : BOOL;  // if TRUE, the instance afterwards gets moved into the copy code (online change)
    eStopper : PMPS.K_Stopper;
    sStopperName : STRING;
END_VAR
Stopper := eStopper;
StopperName := sStopperName;
END_METHOD

END_FUNCTION_BLOCK

// MajorComponents/Stoppers/FB_StopperWatcher
// Relays stopper state and sends a message when stopper state changes.
FUNCTION_BLOCK FB_StopperWatcher
VAR_INPUT
END_VAR
VAR_OUTPUT
END_VAR
VAR_IN_OUT
	stCurrentBP : ST_BeamParams;
END_VAR
VAR
    i_StopperOutLS AT %I* : BOOL;
    i_StopperInLS AT %I* : BOOL;

    q_StopperOUT_Relay AT %Q* : BOOL;
    q_StopperIN_Relay AT %Q* : BOOL;

    Stopper : UINT;
    StopperName : STRING;
	{attribute 'instance-path'}
    {attribute 'noinit'}
    sPath    :    T_MaxString;

    // Logging
    fbLogMsg : FB_LogMessage := (
        eSubSystem := E_Subsystem.MPS);

    rtIn : R_TRIG;
    rtOut : R_TRIG;

	bInit: BOOL := TRUE;
END_VAR

IF bInit THEN
	fbLogMsg.sJson := F_PMPS_JSON(StopperName, sPath, 1000);
	bInit := FALSE;
END_IF


rtIn(CLK := i_StopperInLS);
rtOut(CLK := i_StopperOutLS);

IF rtIn.Q THEN
    fbLogMsg.sMsg := CONCAT(StopperName, ' moved IN');
    fbLogMsg();
ELSIF rtOut.Q THEN
    fbLogMsg.sMsg := CONCAT(StopperName, ' moved OUT');
    fbLogMsg();
END_IF

q_StopperOUT_Relay := i_StopperOutLS;
q_StopperIN_Relay := i_StopperInLS;

// Update current beam parameters
stCurrentBP.aStoppers[Stopper] := i_StopperInLS;

END_FUNCTION_BLOCK

// MajorComponents/Stoppers/FB_LStopper
FUNCTION_BLOCK FB_LStopper EXTENDS FB_StopperWatcher
VAR_INPUT
END_VAR
VAR_OUTPUT
END_VAR
VAR_IN_OUT
END_VAR
VAR
END_VAR

SUPER^(stCurrentBP:=SUPER^.stCurrentBP);

METHOD FB_init : BOOL
VAR_INPUT
    bInitRetains : BOOL; // if TRUE, the retain variables are initialized (warm start / cold start)
    bInCopyCode : BOOL;  // if TRUE, the instance afterwards gets moved into the copy code (online change)
    eStopper : PMPS.L_Stopper;
    sStopperName : STRING;
END_VAR
Stopper := eStopper;
StopperName := sStopperName;
END_METHOD

END_FUNCTION_BLOCK

// MajorComponents/BeamParameterTransitionManager
(*
Implements the procedure for safely transitioning between device states by asserting the correct beam parameters for 
the state *)
FUNCTION_BLOCK BeamParameterTransitionManager
VAR_IN_OUT
    
    fbArbiter    :    FB_Arbiter; //Connect to local arbiter
    
END_VAR
VAR_INPUT
    i_TransitionAssertionID    :    UDINT := 0;
    i_stTransitionAssertion : ST_BeamParams := PMPS_GVL.cstSafeBeam; //Assertion required during transition (always safer than anything inbetween)
    
    i_nRequestedAssertionID    :    UDINT := 0;
    i_stRequestedAssertion    :    ST_BeamParams := PMPS_GVL.cstSafeBeam; //Requested assertion, change whenever
    
    i_xMoving    :    BOOL := FALSE; //Provide rising edge when device begins moving <remove>
    i_xDoneMoving    :    BOOL := FALSE; //Provide rising edge when device is done with a move
    
    stCurrentBeamParameters    :    ST_BeamParams := PMPS_GVL.cstFullBeam; //Connect to current beam parameters
    
END_VAR
VAR_OUTPUT

    q_xTransitionAuthorized    :    BOOL := FALSE; //Rising edge indicating the device is safe to move, use as input to move execute (which requires a rising edge)

END_VAR

VAR
    nTargetAssertionID    :    UDINT := 0;
    stTargetAssertion    :    ST_BeamParams; //Current target assertion
    nCurrentAssertionID    :    UDINT := 0;
    
    xNewBP    :    BOOL;
    xTranBP    :    BOOL;
    xFinalBP    :    BOOL;
    
    eBPTMState : E_BPTMState := Init;
    ePrevState : E_BPTMState := Init;
    
    xEntry : BOOL;
    rTransition : R_TRIG;
    xNewTarget : BOOL;
	
	bTransAssertionFailed : BOOL;
    bFinalAssertionFailed : BOOL;
	
END_VAR


// Execute exit actions before transition back to NewTarget
IF nTargetAssertionID <> i_nRequestedAssertionID THEN
    CASE eBPTMState OF
        //NewTarget:
        WaitingForTransitionAssertion:
            WaitingForTransitionAssertion_EXIT();
        WaitingForFinalAssertion:
            WaitingForFinalAssertion_EXIT();
        Transitioning:
            DeauthorizeTransition();
        //CleaningUp: 
	END_CASE
    
    eBPTMState := E_BPTMState.NewTarget;
    xEntry := eBPTMState <> ePrevState;
    
END_IF



// States
CASE eBPTMState OF
    NewTarget:
        IF xEntry THEN
            NewTarget_ENTRY();
        ELSIF xNewBP THEN
            eBPTMState := E_BPTMState.WaitingForTransitionAssertion;
        ELSE
            SetNewTarget();
        END_IF
            
    WaitingForTransitionAssertion:
        IF xEntry OR bTransAssertionFailed THEN
            AssertTransitionBP();
        ELSIF xTranBP THEN
            WaitingForTransitionAssertion_EXIT();
            eBPTMState := E_BPTMState.WaitingForFinalAssertion;
        ELSE
            WaitingForTransitionAssertion_DO();
        END_IF
        
    WaitingForFinalAssertion:
        IF xEntry OR bFinalAssertionFailed THEN
            AssertFinalBP();
        ELSIF xFinalBP THEN
            WaitingForFinalAssertion_EXIT();
            eBPTMState := E_BPTMState.Transitioning;
        ELSE
            WaitingForFinalAssertion_DO();
        END_IF
        
    Transitioning:
        IF xEntry THEN
            AuthorizeTransition();
        ELSIF i_xDoneMoving THEN
            DeauthorizeTransition();
            eBPTMState := E_BPTMState.CleaningUp;
		END_IF
        
    CleaningUp:
        IF xEntry THEN
            RemoveTransitionAssertion();
		ELSE
			eBPTMState := E_BPTMState.Idle;
		END_IF
END_CASE

xEntry := ePrevState <> eBPTMState;
ePrevState := eBPTMState;

ACTION AssertFinalBP:
//q_stFinalAssertion := stTargetAssertion;

//Clearing previous target parameters
(* This is considered safe at this step as the transition
state beam parameters should always be safer than the
current or target state beam parameters
*)
fbArbiter.RemoveRequest( nCurrentAssertionID );

//Asserting target parameters
bFinalAssertionFailed := NOT fbArbiter.AddRequest(
    nTargetAssertionID,
    stTargetAssertion
);

//Remembering final assertionID for removal later
IF NOT bFinalAssertionFailed THEN
	nCurrentAssertionID := nTargetAssertionID;
END_IF
END_ACTION

ACTION AssertTransitionBP:

bTransAssertionFailed := NOT fbArbiter.AddRequest(
    i_TransitionAssertionID,
    i_stTransitionAssertion
);
END_ACTION

ACTION AuthorizeTransition:
q_xTransitionAuthorized := TRUE;
END_ACTION

ACTION DeauthorizeTransition:
q_xTransitionAuthorized := FALSE;
END_ACTION

ACTION NewTarget_ENTRY:
xNewBP := False;
END_ACTION

ACTION RemoveTransitionAssertion:
//q_stTransitionAssertion := PMPS_GVL.cstFullBeam;

//Removing transition assertion
fbArbiter.RemoveRequest( i_TransitionAssertionID );



//TODO add something to verify removal
END_ACTION

ACTION SetNewTarget:
IF i_nRequestedAssertionID <> 0 AND
    i_nRequestedAssertionID <> PMPS_GVL.EXCLUDED_ASSERTION_ID THEN
    
    stTargetAssertion := i_stRequestedAssertion;
    nTargetAssertionID := i_nRequestedAssertionID;
    xNewBP := TRUE;
END_IF
END_ACTION

ACTION WaitingForFinalAssertion_DO:
//Final Assertion Verification

xFinalBP := F_SafeBPCompare(stCurrentBeamParameters, stTargetAssertion) AND
    fbArbiter.CheckRequest( i_nRequestedAssertionID);;
END_ACTION

ACTION WaitingForFinalAssertion_EXIT:
//Set this bool false so we can get a rising edge on the next try
xFinalBP := FALSE;
PMPS_GVL.SuccessfulPreemption := PMPS_GVL.SuccessfulPreemption + 1;
END_ACTION

ACTION WaitingForTransitionAssertion_DO:
//Transition Assertion Verification
xTranBP    := F_SafeBPCompare(stCurrentBeamParameters, i_stTransitionAssertion) AND
    fbArbiter.CheckRequest(i_TransitionAssertionID);
END_ACTION

ACTION WaitingForTransitionAssertion_EXIT:
xTranBP := FALSE;
PMPS_GVL.SuccessfulPreemption := PMPS_GVL.SuccessfulPreemption + 1;
END_ACTION

END_FUNCTION_BLOCK

